LIN {X -0.032,Y -439.695,Z 1064.574,A 0.000,B 0.000,C 90.000,E1 103.300} C_DIS
LIN {X -0.146,Y -459.814,Z 1064.563,A 0.000,B 0.000,C 90.000,E1 101.299} C_DIS
LIN {X 0.195,Y -467.473,Z 1064.559,A 0.000,B 0.000,C 90.000,E1 100.546} C_DIS
LIN {X 0.213,Y -469.559,Z 1064.557,A 0.000,B 0.000,C 90.000,E1 100.310} C_DIS
LIN {X 0.062,Y -471.262,Z 1064.556,A 0.000,B 0.000,C 90.000,E1 100.074} C_DIS
LIN {X -0.172,Y -472.541,Z 1064.555,A 0.000,B 0.000,C 90.000,E1 99.849} C_DIS
LIN {X 0.011,Y -474.126,Z 1064.552,A 0.000,B 0.000,C 90.000,E1 99.321} C_DIS
LIN {X 0.125,Y -474.657,Z 1064.549,A 0.000,B 0.000,C 90.000,E1 98.803} C_DIS
LIN {X -0.219,Y -474.225,Z 1064.546,A 0.000,B 0.000,C 90.000,E1 98.341} C_DIS
LIN {X -0.024,Y -472.767,Z 1064.543,A 0.000,B 0.000,C 90.000,E1 97.814} C_DIS
LIN {X -0.227,Y -471.579,Z 1064.542,A 0.000,B 0.000,C 90.000,E1 97.587} C_DIS
LIN {X -0.105,Y -468.181,Z 1064.539,A 0.000,B 0.000,C 90.000,E1 97.068} C_DIS
LIN {X -0.042,Y -455.689,Z 1064.529,A 0.000,B 0.000,C 90.000,E1 95.277} C_DIS
LIN {X -0.126,Y -441.483,Z 1064.518,A 0.000,B 0.000,C 90.000,E1 93.212} C_DIS
LIN {X -0.111,Y -423.738,Z 1064.501,A 0.000,B 0.000,C 90.000,E1 90.286} C_DIS
LIN {X 0.172,Y -407.307,Z 1064.485,A 0.000,B 0.000,C 90.000,E1 87.249} C_DIS
LIN {X 0.158,Y -398.335,Z 1064.476,A 0.000,B 0.000,C 90.000,E1 85.584} C_DIS
LIN {X 0.025,Y -389.176,Z 1064.466,A 0.000,B 0.000,C 90.000,E1 83.913} C_DIS
LIN {X 0.131,Y -378.261,Z 1064.455,A 0.000,B 0.000,C 90.000,E1 81.894} C_DIS
LIN {X 0.126,Y -370.259,Z 1064.447,A 0.000,B 0.000,C 90.000,E1 80.443} C_DIS
LIN {X -0.030,Y -360.352,Z 1064.437,A 0.000,B 0.000,C 90.000,E1 78.701} C_DIS
LIN {X 0.062,Y -348.682,Z 1064.426,A 0.000,B 0.000,C 90.000,E1 76.589} C_DIS
LIN {X -0.132,Y -333.953,Z 1064.410,A 0.000,B 0.000,C 90.000,E1 73.866} C_DIS
LIN {X -0.123,Y -319.754,Z 1064.395,A 0.000,B 0.000,C 90.000,E1 71.040} C_DIS
LIN {X 0.015,Y -304.809,Z 1064.377,A 0.000,B 0.000,C 90.000,E1 67.794} C_DIS
LIN {X 0.035,Y -293.366,Z 1064.362,A 0.000,B 0.000,C 90.000,E1 65.153} C_DIS
LIN {X 0.087,Y -284.911,Z 1064.351,A 0.000,B 0.000,C 90.000,E1 63.127} C_DIS
LIN {X -0.007,Y -273.876,Z 1064.336,A 0.000,B 0.000,C 90.000,E1 60.411} C_DIS
LIN {X 0.165,Y -263.096,Z 1064.320,A 0.000,B 0.000,C 90.000,E1 57.582} C_DIS
LIN {X 0.021,Y -251.353,Z 1064.302,A 0.000,B 0.000,C 90.000,E1 54.402} C_DIS
LIN {X -0.006,Y -241.398,Z 1064.286,A 0.000,B 0.000,C 90.000,E1 51.492} C_DIS
LIN {X -0.088,Y -230.859,Z 1064.267,A 0.000,B 0.000,C 90.000,E1 48.162} C_DIS
LIN {X 0.020,Y -221.065,Z 1064.248,A 0.000,B 0.000,C 90.000,E1 44.717} C_DIS
LIN {X -0.019,Y -212.891,Z 1064.231,A 0.000,B 0.000,C 90.000,E1 41.634} C_DIS
LIN {X 0.064,Y -205.107,Z 1064.214,A 0.000,B 0.000,C 90.000,E1 38.463} C_DIS
LIN {X -0.106,Y -197.961,Z 1064.196,A 0.000,B 0.000,C 90.000,E1 35.311} C_DIS
LIN {X 0.082,Y -191.433,Z 1064.178,A 0.000,B 0.000,C 90.000,E1 32.005} C_DIS
LIN {X -0.035,Y -185.633,Z 1064.160,A 0.000,B 0.000,C 90.000,E1 28.743} C_DIS
LIN {X -0.062,Y -180.529,Z 1064.141,A 0.000,B 0.000,C 90.000,E1 25.412} C_DIS
LIN {X -0.037,Y -176.142,Z 1064.122,A 0.000,B 0.000,C 90.000,E1 22.025} C_DIS
LIN {X 0.006,Y -172.503,Z 1064.103,A 0.000,B 0.000,C 90.000,E1 18.598} C_DIS
LIN {X -0.017,Y -168.891,Z 1064.079,A 0.000,B 0.000,C 90.000,E1 14.300} C_DIS
LIN {X -0.035,Y -165.957,Z 1064.050,A 0.000,B 0.000,C 90.000,E1 9.095} C_DIS
LIN {X 0.021,Y -164.114,Z 1064.007,A 0.000,B 0.000,C 90.000,E1 1.203} C_DIS
LIN {X -0.010,Y -165.807,Z 1063.958,A 0.000,B 0.000,C 90.000,E1 352.527} C_DIS
LIN {X -0.018,Y -168.701,Z 1063.929,A 0.000,B 0.000,C 90.000,E1 347.297} C_DIS
LIN {X 0.004,Y -172.281,Z 1063.905,A 0.000,B 0.000,C 90.000,E1 342.960} C_DIS
LIN {X 0.023,Y -175.889,Z 1063.886,A 0.000,B 0.000,C 90.000,E1 339.518} C_DIS
LIN {X 0.053,Y -180.218,Z 1063.867,A 0.000,B 0.000,C 90.000,E1 336.102} C_DIS
LIN {X 0.009,Y -185.294,Z 1063.849,A 0.000,B 0.000,C 90.000,E1 332.743} C_DIS
LIN {X 0.012,Y -191.186,Z 1063.830,A 0.000,B 0.000,C 90.000,E1 329.410} C_DIS
LIN {X -0.034,Y -197.896,Z 1063.812,A 0.000,B 0.000,C 90.000,E1 326.135} C_DIS
LIN {X -0.009,Y -205.317,Z 1063.794,A 0.000,B 0.000,C 90.000,E1 322.889} C_DIS
LIN {X 0.047,Y -214.515,Z 1063.774,A 0.000,B 0.000,C 90.000,E1 319.299} C_DIS
LIN {X -0.076,Y -223.380,Z 1063.757,A 0.000,B 0.000,C 90.000,E1 316.215} C_DIS
LIN {X -0.097,Y -231.825,Z 1063.742,A 0.000,B 0.000,C 90.000,E1 313.542} C_DIS
LIN {X -0.099,Y -242.772,Z 1063.725,A 0.000,B 0.000,C 90.000,E1 310.539} C_DIS
LIN {X 0.024,Y -250.496,Z 1063.715,A 0.000,B 0.000,C 90.000,E1 308.669} C_DIS
LIN {X -0.007,Y -260.943,Z 1063.703,A 0.000,B 0.000,C 90.000,E1 306.503} C_DIS
LIN {X 0.163,Y -278.361,Z 1063.685,A 0.000,B 0.000,C 90.000,E1 303.293} C_DIS
LIN {X 0.013,Y -294.989,Z 1063.670,A 0.000,B 0.000,C 90.000,E1 300.590} C_DIS
LIN {X -0.175,Y -312.721,Z 1063.655,A 0.000,B 0.000,C 90.000,E1 297.975} C_DIS
LIN {X -0.152,Y -329.507,Z 1063.643,A 0.000,B 0.000,C 90.000,E1 295.720} C_DIS
LIN {X -0.105,Y -339.902,Z 1063.636,A 0.000,B 0.000,C 90.000,E1 294.463} C_DIS
LIN {X -0.113,Y -355.907,Z 1063.626,A 0.000,B 0.000,C 90.000,E1 292.770} C_DIS
LIN {X 0.102,Y -375.164,Z 1063.616,A 0.000,B 0.000,C 90.000,E1 290.918} C_DIS
LIN {X 0.090,Y -394.606,Z 1063.607,A 0.000,B 0.000,C 90.000,E1 289.214} C_DIS
LIN {X -0.133,Y -405.562,Z 1063.602,A 0.000,B 0.000,C 90.000,E1 288.308} C_DIS
LIN {X 0.077,Y -416.195,Z 1063.596,A 0.000,B 0.000,C 90.000,E1 287.330} C_DIS
LIN {X 0.042,Y -423.799,Z 1063.592,A 0.000,B 0.000,C 90.000,E1 286.622} C_DIS
LIN {X 0.136,Y -430.980,Z 1063.588,A 0.000,B 0.000,C 90.000,E1 285.898} C_DIS
LIN {X -0.129,Y -440.679,Z 1063.583,A 0.000,B 0.000,C 90.000,E1 284.898} C_DIS
LIN {X 0.191,Y -447.662,Z 1063.578,A 0.000,B 0.000,C 90.000,E1 284.064} C_DIS
LIN {X 0.035,Y -454.176,Z 1063.574,A 0.000,B 0.000,C 90.000,E1 283.300} C_DIS
LIN {X -0.074,Y -459.997,Z 1063.570,A 0.000,B 0.000,C 90.000,E1 282.535} C_DIS
LIN {X -0.127,Y -465.162,Z 1063.565,A 0.000,B 0.000,C 90.000,E1 281.771} C_DIS
LIN {X -0.143,Y -469.654,Z 1063.561,A 0.000,B 0.000,C 90.000,E1 281.007} C_DIS
LIN {X -0.205,Y -473.432,Z 1063.557,A 0.000,B 0.000,C 90.000,E1 280.254} C_DIS
LIN {X -0.233,Y -476.636,Z 1063.553,A 0.000,B 0.000,C 90.000,E1 279.500} C_DIS
LIN {X -0.026,Y -478.476,Z 1063.550,A 0.000,B 0.000,C 90.000,E1 278.973} C_DIS
LIN {X 0.114,Y -480.089,Z 1063.547,A 0.000,B 0.000,C 90.000,E1 278.454} C_DIS
LIN {X 0.017,Y -482.687,Z 1063.542,A 0.000,B 0.000,C 90.000,E1 277.466} C_DIS
LIN {X 0.187,Y -483.768,Z 1063.539,A 0.000,B 0.000,C 90.000,E1 276.947} C_DIS
LIN {X -0.116,Y -484.581,Z 1063.536,A 0.000,B 0.000,C 90.000,E1 276.486} C_DIS
LIN {X 0.067,Y -485.137,Z 1063.533,A 0.000,B 0.000,C 90.000,E1 275.967} C_DIS
LIN {X 0.209,Y -485.234,Z 1063.530,A 0.000,B 0.000,C 90.000,E1 275.454} C_DIS
LIN {X -0.080,Y -484.976,Z 1063.528,A 0.000,B 0.000,C 90.000,E1 274.992} C_DIS
LIN {X 0.112,Y -484.243,Z 1063.525,A 0.000,B 0.000,C 90.000,E1 274.473} C_DIS
LIN {X -0.181,Y -482.986,Z 1063.522,A 0.000,B 0.000,C 90.000,E1 274.012} C_DIS
LIN {X -0.031,Y -481.115,Z 1063.519,A 0.000,B 0.000,C 90.000,E1 273.498} C_DIS
LIN {X 0.141,Y -478.649,Z 1063.517,A 0.000,B 0.000,C 90.000,E1 272.980} C_DIS
LIN {X -0.206,Y -475.363,Z 1063.514,A 0.000,B 0.000,C 90.000,E1 272.522} C_DIS
LIN {X -0.089,Y -471.247,Z 1063.511,A 0.000,B 0.000,C 90.000,E1 272.007} C_DIS
LIN {X 0.020,Y -466.048,Z 1063.508,A 0.000,B 0.000,C 90.000,E1 271.489} C_DIS
LIN {X -0.096,Y -460.287,Z 1063.506,A 0.000,B 0.000,C 90.000,E1 271.031} C_DIS
LIN {X 0.167,Y -454.105,Z 1063.503,A 0.000,B 0.000,C 90.000,E1 270.573} C_DIS
LIN {X -0.046,Y -447.420,Z 1063.501,A 0.000,B 0.000,C 90.000,E1 270.229} C_DIS
LIN {X -0.220,Y -440.237,Z 1063.500,A 0.000,B 0.000,C 90.000,E1 269.943} C_DIS
LIN {X 0.089,Y -432.502,Z 1063.498,A 0.000,B 0.000,C 90.000,E1 269.656} C_DIS
LIN {X 0.000,Y -424.409,Z 1063.497,A 0.000,B 0.000,C 90.000,E1 269.484} C_DIS
LIN {X -0.129,Y -415.458,Z 1063.496,A 0.000,B 0.000,C 90.000,E1 269.370} C_DIS
LIN {X 0.032,Y -406.189,Z 1063.496,A 0.000,B 0.000,C 90.000,E1 269.255} C_DIS
LIN {X 0.039,Y -395.853,Z 1063.496,A 0.000,B 0.000,C 90.000,E1 269.198} C_DIS
LIN {X -0.012,Y -181.363,Z 1063.495,A 0.000,B 0.000,C 90.000,E1 269.198} C_DIS
LIN {X 0.045,Y -180.907,Z 1063.475,A 0.000,B 0.000,C 90.000,E1 265.469} C_DIS
LIN {X -0.078,Y -180.743,Z 1063.470,A 0.000,B 0.000,C 90.000,E1 264.666} C_DIS
LIN {X 0.023,Y -178.834,Z 1063.442,A 0.000,B 0.000,C 90.000,E1 259.567} C_DIS
LIN {X 0.057,Y -175.878,Z 1063.414,A 0.000,B 0.000,C 90.000,E1 254.464} C_DIS
LIN {X -0.006,Y -174.538,Z 1063.404,A 0.000,B 0.000,C 90.000,E1 252.779} C_DIS
LIN {X 0.087,Y -171.523,Z 1063.380,A 0.000,B 0.000,C 90.000,E1 248.465} C_DIS
LIN {X 0.072,Y -167.749,Z 1063.357,A 0.000,B 0.000,C 90.000,E1 244.152} C_DIS
LIN {X 0.011,Y -166.451,Z 1063.347,A 0.000,B 0.000,C 90.000,E1 242.436} C_DIS
LIN {X 0.001,Y -163.168,Z 1063.328,A 0.000,B 0.000,C 90.000,E1 238.948} C_DIS
LIN {X 0.050,Y -161.126,Z 1063.313,A 0.000,B 0.000,C 90.000,E1 236.294} C_DIS
LIN {X -0.047,Y -157.148,Z 1063.288,A 0.000,B 0.000,C 90.000,E1 231.904} C_DIS
LIN {X -0.024,Y -155.881,Z 1063.278,A 0.000,B 0.000,C 90.000,E1 230.114} C_DIS
LIN {X -0.065,Y -152.132,Z 1063.253,A 0.000,B 0.000,C 90.000,E1 225.648} C_DIS
LIN {X -0.045,Y -150.381,Z 1063.238,A 0.000,B 0.000,C 90.000,E1 222.933} C_DIS
LIN {X -0.021,Y -147.114,Z 1063.213,A 0.000,B 0.000,C 90.000,E1 218.382} C_DIS
LIN {X -0.029,Y -145.680,Z 1063.198,A 0.000,B 0.000,C 90.000,E1 215.644} C_DIS
LIN {X -0.031,Y -143.062,Z 1063.172,A 0.000,B 0.000,C 90.000,E1 211.052} C_DIS
LIN {X 0.026,Y -141.683,Z 1063.152,A 0.000,B 0.000,C 90.000,E1 207.334} C_DIS
LIN {X 0.005,Y -139.458,Z 1063.116,A 0.000,B 0.000,C 90.000,E1 200.844} C_DIS
LIN {X 0.056,Y -139.192,Z 1063.105,A 0.000,B 0.000,C 90.000,E1 198.960} C_DIS
LIN {X -0.057,Y -138.325,Z 1063.054,A 0.000,B 0.000,C 90.000,E1 189.670} C_DIS
LIN {X -0.053,Y -139.455,Z 1063.007,A 0.000,B 0.000,C 90.000,E1 181.260} C_DIS
LIN {X 0.027,Y -141.003,Z 1062.976,A 0.000,B 0.000,C 90.000,E1 175.641} C_DIS
LIN {X -0.023,Y -142.757,Z 1062.955,A 0.000,B 0.000,C 90.000,E1 171.951} C_DIS
LIN {X -0.068,Y -145.160,Z 1062.930,A 0.000,B 0.000,C 90.000,E1 167.353} C_DIS
LIN {X -0.076,Y -147.782,Z 1062.909,A 0.000,B 0.000,C 90.000,E1 163.685} C_DIS
LIN {X 0.003,Y -150.461,Z 1062.889,A 0.000,B 0.000,C 90.000,E1 160.007} C_DIS
LIN {X 0.079,Y -153.912,Z 1062.869,A 0.000,B 0.000,C 90.000,E1 156.357} C_DIS
LIN {X 0.003,Y -157.323,Z 1062.849,A 0.000,B 0.000,C 90.000,E1 152.794} C_DIS
LIN {X 0.087,Y -161.511,Z 1062.829,A 0.000,B 0.000,C 90.000,E1 149.203} C_DIS
LIN {X -0.036,Y -165.710,Z 1062.809,A 0.000,B 0.000,C 90.000,E1 145.722} C_DIS
LIN {X 0.089,Y -170.656,Z 1062.790,A 0.000,B 0.000,C 90.000,E1 142.190} C_DIS
LIN {X 0.002,Y -175.533,Z 1062.771,A 0.000,B 0.000,C 90.000,E1 138.771} C_DIS
LIN {X -0.004,Y -181.152,Z 1062.752,A 0.000,B 0.000,C 90.000,E1 135.364} C_DIS
LIN {X -0.007,Y -186.605,Z 1062.733,A 0.000,B 0.000,C 90.000,E1 132.000} C_DIS
LIN {X 0.063,Y -191.214,Z 1062.719,A 0.000,B 0.000,C 90.000,E1 129.483} C_DIS
LIN {X -0.009,Y -197.425,Z 1062.700,A 0.000,B 0.000,C 90.000,E1 126.011} C_DIS
LIN {X -0.052,Y -198.581,Z 1062.697,A 0.000,B 0.000,C 90.000,E1 125.438} C_DIS
LIN {X -0.114,Y -305.000,Z 1062.697,A 0.000,B 0.000,C 90.000,E1 125.438} C_DIS
LIN {X 0.033,Y -306.362,Z 1062.697,A 0.000,B 0.000,C 90.000,E1 125.391} C_DIS
LIN {X -0.186,Y -309.700,Z 1062.696,A 0.000,B 0.000,C 90.000,E1 125.311} C_DIS
LIN {X 0.137,Y -312.965,Z 1062.695,A 0.000,B 0.000,C 90.000,E1 125.025} C_DIS
LIN {X 0.124,Y -316.653,Z 1062.692,A 0.000,B 0.000,C 90.000,E1 124.612} C_DIS
LIN {X 0.011,Y -318.561,Z 1062.691,A 0.000,B 0.000,C 90.000,E1 124.326} C_DIS
LIN {X 0.161,Y -320.060,Z 1062.689,A 0.000,B 0.000,C 90.000,E1 123.992} C_DIS
LIN {X -0.136,Y -323.460,Z 1062.684,A 0.000,B 0.000,C 90.000,E1 123.086} C_DIS
LIN {X 0.070,Y -333.960,Z 1062.668,A 0.000,B 0.000,C 90.000,E1 120.207} C_DIS
LIN {X -0.043,Y -345.811,Z 1062.652,A 0.000,B 0.000,C 90.000,E1 117.436} C_DIS
LIN {X -0.005,Y -359.122,Z 1062.637,A 0.000,B 0.000,C 90.000,E1 114.695} C_DIS
LIN {X -0.119,Y -372.270,Z 1062.624,A 0.000,B 0.000,C 90.000,E1 112.333} C_DIS
LIN {X -0.042,Y -386.756,Z 1062.611,A 0.000,B 0.000,C 90.000,E1 109.993} C_DIS
LIN {X 0.138,Y -402.680,Z 1062.598,A 0.000,B 0.000,C 90.000,E1 107.692} C_DIS
LIN {X 0.088,Y -420.157,Z 1062.586,A 0.000,B 0.000,C 90.000,E1 105.481} C_DIS
LIN {X -0.155,Y -439.292,Z 1062.574,A 0.000,B 0.000,C 90.000,E1 103.355} C_DIS
LIN {X 0.146,Y -459.401,Z 1062.563,A 0.000,B 0.000,C 90.000,E1 101.299} C_DIS
LIN {X 0.023,Y -467.071,Z 1062.559,A 0.000,B 0.000,C 90.000,E1 100.602} C_DIS
LIN {X 0.036,Y -469.257,Z 1062.558,A 0.000,B 0.000,C 90.000,E1 100.366} C_DIS
LIN {X -0.199,Y -471.030,Z 1062.556,A 0.000,B 0.000,C 90.000,E1 100.141} C_DIS
LIN {X 0.113,Y -472.363,Z 1062.555,A 0.000,B 0.000,C 90.000,E1 99.849} C_DIS
LIN {X -0.172,Y -474.028,Z 1062.552,A 0.000,B 0.000,C 90.000,E1 99.378} C_DIS
LIN {X -0.062,Y -474.628,Z 1062.549,A 0.000,B 0.000,C 90.000,E1 98.859} C_DIS
LIN {X 0.063,Y -474.263,Z 1062.546,A 0.000,B 0.000,C 90.000,E1 98.341} C_DIS
LIN {X -0.211,Y -472.881,Z 1062.544,A 0.000,B 0.000,C 90.000,E1 97.871} C_DIS
LIN {X 0.054,Y -471.740,Z 1062.542,A 0.000,B 0.000,C 90.000,E1 97.587} C_DIS
LIN {X -0.085,Y -470.219,Z 1062.541,A 0.000,B 0.000,C 90.000,E1 97.352} C_DIS
LIN {X 0.234,Y -455.909,Z 1062.530,A 0.000,B 0.000,C 90.000,E1 95.277} C_DIS
LIN {X -0.091,Y -440.013,Z 1062.516,A 0.000,B 0.000,C 90.000,E1 92.980} C_DIS
LIN {X -0.018,Y -420.855,Z 1062.499,A 0.000,B 0.000,C 90.000,E1 89.771} C_DIS
LIN {X 0.029,Y -407.518,Z 1062.485,A 0.000,B 0.000,C 90.000,E1 87.306} C_DIS
LIN {X 0.023,Y -398.552,Z 1062.476,A 0.000,B 0.000,C 90.000,E1 85.641} C_DIS
LIN {X -0.102,Y -389.400,Z 1062.466,A 0.000,B 0.000,C 90.000,E1 83.970} C_DIS
LIN {X 0.014,Y -378.487,Z 1062.455,A 0.000,B 0.000,C 90.000,E1 81.951} C_DIS
LIN {X 0.016,Y -370.516,Z 1062.447,A 0.000,B 0.000,C 90.000,E1 80.500} C_DIS
LIN {X -0.131,Y -360.565,Z 1062.437,A 0.000,B 0.000,C 90.000,E1 78.757} C_DIS
LIN {X -0.029,Y -348.903,Z 1062.426,A 0.000,B 0.000,C 90.000,E1 76.645} C_DIS
LIN {X 0.113,Y -334.198,Z 1062.411,A 0.000,B 0.000,C 90.000,E1 73.866} C_DIS
LIN {X 0.117,Y -319.964,Z 1062.395,A 0.000,B 0.000,C 90.000,E1 71.040} C_DIS
LIN {X -0.032,Y -305.005,Z 1062.377,A 0.000,B 0.000,C 90.000,E1 67.847} C_DIS
LIN {X -0.124,Y -293.541,Z 1062.362,A 0.000,B 0.000,C 90.000,E1 65.229} C_DIS
LIN {X -0.092,Y -283.663,Z 1062.349,A 0.000,B 0.000,C 90.000,E1 62.871} C_DIS
LIN {X -0.077,Y -272.652,Z 1062.334,A 0.000,B 0.000,C 90.000,E1 60.127} C_DIS
LIN {X -0.066,Y -261.880,Z 1062.318,A 0.000,B 0.000,C 90.000,E1 57.327} C_DIS
LIN {X -0.099,Y -250.180,Z 1062.301,A 0.000,B 0.000,C 90.000,E1 54.116} C_DIS
LIN {X -0.001,Y -240.219,Z 1062.284,A 0.000,B 0.000,C 90.000,E1 51.170} C_DIS
LIN {X 0.067,Y -229.739,Z 1062.266,A 0.000,B 0.000,C 90.000,E1 47.796} C_DIS
LIN {X 0.053,Y -221.070,Z 1062.249,A 0.000,B 0.000,C 90.000,E1 44.757} C_DIS
LIN {X 0.003,Y -212.870,Z 1062.232,A 0.000,B 0.000,C 90.000,E1 41.676} C_DIS
LIN {X -0.051,Y -205.075,Z 1062.214,A 0.000,B 0.000,C 90.000,E1 38.543} C_DIS
LIN {X 0.060,Y -197.919,Z 1062.196,A 0.000,B 0.000,C 90.000,E1 35.311} C_DIS
LIN {X -0.021,Y -191.371,Z 1062.178,A 0.000,B 0.000,C 90.000,E1 32.084} C_DIS
LIN {X 0.030,Y -185.550,Z 1062.160,A 0.000,B 0.000,C 90.000,E1 28.771} C_DIS
LIN {X -0.078,Y -180.434,Z 1062.141,A 0.000,B 0.000,C 90.000,E1 25.463} C_DIS
LIN {X -0.059,Y -176.029,Z 1062.123,A 0.000,B 0.000,C 90.000,E1 22.078} C_DIS
LIN {X -0.022,Y -172.389,Z 1062.104,A 0.000,B 0.000,C 90.000,E1 18.652} C_DIS
LIN {X -0.051,Y -168.752,Z 1062.080,A 0.000,B 0.000,C 90.000,E1 14.356} C_DIS
LIN {X -0.062,Y -166.194,Z 1062.056,A 0.000,B 0.000,C 90.000,E1 10.018} C_DIS
LIN {X 0.067,Y -164.072,Z 1062.017,A 0.000,B 0.000,C 90.000,E1 2.980} C_DIS
LIN {X 0.004,Y -165.293,Z 1061.963,A 0.000,B 0.000,C 90.000,E1 353.394} C_DIS
LIN {X -0.048,Y -167.974,Z 1061.934,A 0.000,B 0.000,C 90.000,E1 348.173} C_DIS
LIN {X 0.073,Y -171.333,Z 1061.910,A 0.000,B 0.000,C 90.000,E1 343.795} C_DIS
LIN {X 0.017,Y -174.773,Z 1061.891,A 0.000,B 0.000,C 90.000,E1 340.369} C_DIS
LIN {X -0.049,Y -178.917,Z 1061.872,A 0.000,B 0.000,C 90.000,E1 336.975} C_DIS
LIN {X -0.040,Y -183.833,Z 1061.853,A 0.000,B 0.000,C 90.000,E1 333.589} C_DIS
LIN {X -0.076,Y -189.535,Z 1061.835,A 0.000,B 0.000,C 90.000,E1 330.255} C_DIS
LIN {X 0.062,Y -196.027,Z 1061.816,A 0.000,B 0.000,C 90.000,E1 326.914} C_DIS
LIN {X -0.082,Y -203.297,Z 1061.798,A 0.000,B 0.000,C 90.000,E1 323.703} C_DIS
LIN {X 0.004,Y -211.273,Z 1061.780,A 0.000,B 0.000,C 90.000,E1 320.481} C_DIS
LIN {X 0.131,Y -219.857,Z 1061.763,A 0.000,B 0.000,C 90.000,E1 317.310} C_DIS
LIN {X -0.025,Y -229.199,Z 1061.746,A 0.000,B 0.000,C 90.000,E1 314.271} C_DIS
LIN {X 0.070,Y -239.800,Z 1061.729,A 0.000,B 0.000,C 90.000,E1 311.229} C_DIS
LIN {X -0.040,Y -247.155,Z 1061.719,A 0.000,B 0.000,C 90.000,E1 309.402} C_DIS
LIN {X -0.139,Y -257.230,Z 1061.707,A 0.000,B 0.000,C 90.000,E1 307.237} C_DIS
LIN {X 0.080,Y -270.354,Z 1061.693,A 0.000,B 0.000,C 90.000,E1 304.692} C_DIS
LIN {X 0.000,Y -288.580,Z 1061.676,A 0.000,B 0.000,C 90.000,E1 301.592} C_DIS
LIN {X 0.064,Y -305.895,Z 1061.661,A 0.000,B 0.000,C 90.000,E1 298.899} C_DIS
LIN {X 0.100,Y -327.053,Z 1061.644,A 0.000,B 0.000,C 90.000,E1 295.976} C_DIS
LIN {X -0.186,Y -340.026,Z 1061.636,A 0.000,B 0.000,C 90.000,E1 294.463} C_DIS
LIN {X -0.037,Y -353.504,Z 1061.628,A 0.000,B 0.000,C 90.000,E1 293.003} C_DIS
LIN {X -0.079,Y -372.970,Z 1061.617,A 0.000,B 0.000,C 90.000,E1 291.153} C_DIS
LIN {X -0.145,Y -392.379,Z 1061.608,A 0.000,B 0.000,C 90.000,E1 289.450} C_DIS
LIN {X 0.071,Y -406.153,Z 1061.601,A 0.000,B 0.000,C 90.000,E1 288.236} C_DIS
LIN {X 0.119,Y -416.781,Z 1061.596,A 0.000,B 0.000,C 90.000,E1 287.275} C_DIS
LIN {X 0.011,Y -424.440,Z 1061.592,A 0.000,B 0.000,C 90.000,E1 286.567} C_DIS
LIN {X -0.179,Y -431.921,Z 1061.588,A 0.000,B 0.000,C 90.000,E1 285.843} C_DIS
LIN {X 0.008,Y -441.656,Z 1061.582,A 0.000,B 0.000,C 90.000,E1 284.773} C_DIS
LIN {X -0.211,Y -448.606,Z 1061.578,A 0.000,B 0.000,C 90.000,E1 284.008} C_DIS
LIN {X 0.183,Y -454.997,Z 1061.573,A 0.000,B 0.000,C 90.000,E1 283.175} C_DIS
LIN {X 0.081,Y -460.728,Z 1061.569,A 0.000,B 0.000,C 90.000,E1 282.411} C_DIS
LIN {X -0.063,Y -465.811,Z 1061.565,A 0.000,B 0.000,C 90.000,E1 281.658} C_DIS
LIN {X -0.071,Y -470.235,Z 1061.560,A 0.000,B 0.000,C 90.000,E1 280.894} C_DIS
LIN {X -0.124,Y -473.954,Z 1061.556,A 0.000,B 0.000,C 90.000,E1 280.141} C_DIS
LIN {X -0.066,Y -477.123,Z 1061.552,A 0.000,B 0.000,C 90.000,E1 279.378} C_DIS
LIN {X 0.068,Y -478.914,Z 1061.549,A 0.000,B 0.000,C 90.000,E1 278.859} C_DIS
LIN {X 0.212,Y -480.495,Z 1061.547,A 0.000,B 0.000,C 90.000,E1 278.341} C_DIS
LIN {X 0.122,Y -483.081,Z 1061.541,A 0.000,B 0.000,C 90.000,E1 277.352} C_DIS
LIN {X -0.185,Y -484.106,Z 1061.538,A 0.000,B 0.000,C 90.000,E1 276.891} C_DIS
LIN {X -0.005,Y -484.903,Z 1061.535,A 0.000,B 0.000,C 90.000,E1 276.372} C_DIS
LIN {X 0.182,Y -485.384,Z 1061.533,A 0.000,B 0.000,C 90.000,E1 275.853} C_DIS
LIN {X -0.111,Y -485.441,Z 1061.530,A 0.000,B 0.000,C 90.000,E1 275.391} C_DIS
LIN {X 0.041,Y -485.093,Z 1061.527,A 0.000,B 0.000,C 90.000,E1 274.878} C_DIS
LIN {X 0.234,Y -484.238,Z 1061.524,A 0.000,B 0.000,C 90.000,E1 274.359} C_DIS
LIN {X -0.059,Y -482.885,Z 1061.522,A 0.000,B 0.000,C 90.000,E1 273.898} C_DIS
LIN {X 0.092,Y -480.924,Z 1061.519,A 0.000,B 0.000,C 90.000,E1 273.383} C_DIS
LIN {X -0.214,Y -478.285,Z 1061.516,A 0.000,B 0.000,C 90.000,E1 272.922} C_DIS
LIN {X -0.086,Y -474.868,Z 1061.513,A 0.000,B 0.000,C 90.000,E1 272.407} C_DIS
LIN {X 0.028,Y -470.537,Z 1061.510,A 0.000,B 0.000,C 90.000,E1 271.892} C_DIS
LIN {X 0.131,Y -465.160,Z 1061.508,A 0.000,B 0.000,C 90.000,E1 271.375} C_DIS
LIN {X 0.093,Y -459.290,Z 1061.505,A 0.000,B 0.000,C 90.000,E1 270.917} C_DIS
LIN {X -0.030,Y -453.038,Z 1061.503,A 0.000,B 0.000,C 90.000,E1 270.516} C_DIS
LIN {X -0.146,Y -446.382,Z 1061.501,A 0.000,B 0.000,C 90.000,E1 270.172} C_DIS
LIN {X 0.184,Y -439.078,Z 1061.499,A 0.000,B 0.000,C 90.000,E1 269.828} C_DIS
LIN {X 0.145,Y -435.601,Z 1061.499,A 0.000,B 0.000,C 90.000,E1 269.714} C_DIS
LIN {X -0.086,Y -427.543,Z 1061.497,A 0.000,B 0.000,C 90.000,E1 269.542} C_DIS
LIN {X 0.110,Y -419.418,Z 1061.497,A 0.000,B 0.000,C 90.000,E1 269.370} C_DIS
LIN {X 0.168,Y -410.058,Z 1061.496,A 0.000,B 0.000,C 90.000,E1 269.255} C_DIS
LIN {X -0.054,Y -395.709,Z 1061.495,A 0.000,B 0.000,C 90.000,E1 269.198} C_DIS
LIN {X -0.053,Y -181.361,Z 1061.495,A 0.000,B 0.000,C 90.000,E1 269.198} C_DIS
LIN {X -0.023,Y -180.907,Z 1061.475,A 0.000,B 0.000,C 90.000,E1 265.469} C_DIS
LIN {X 0.034,Y -180.733,Z 1061.470,A 0.000,B 0.000,C 90.000,E1 264.609} C_DIS
LIN {X -0.045,Y -178.823,Z 1061.442,A 0.000,B 0.000,C 90.000,E1 259.567} C_DIS
LIN {X 0.037,Y -175.867,Z 1061.414,A 0.000,B 0.000,C 90.000,E1 254.448} C_DIS
LIN {X 0.032,Y -173.837,Z 1061.399,A 0.000,B 0.000,C 90.000,E1 251.891} C_DIS
LIN {X 0.020,Y -171.504,Z 1061.380,A 0.000,B 0.000,C 90.000,E1 248.465} C_DIS
LIN {X 0.007,Y -167.733,Z 1061.356,A 0.000,B 0.000,C 90.000,E1 244.152} C_DIS
LIN {X 0.022,Y -166.429,Z 1061.347,A 0.000,B 0.000,C 90.000,E1 242.410} C_DIS
LIN {X 0.021,Y -163.149,Z 1061.327,A 0.000,B 0.000,C 90.000,E1 238.918} C_DIS
LIN {X -0.013,Y -161.105,Z 1061.313,A 0.000,B 0.000,C 90.000,E1 236.294} C_DIS
LIN {X -0.030,Y -157.831,Z 1061.293,A 0.000,B 0.000,C 90.000,E1 232.763} C_DIS
LIN {X 0.033,Y -155.864,Z 1061.278,A 0.000,B 0.000,C 90.000,E1 230.070} C_DIS
LIN {X 0.088,Y -152.114,Z 1061.253,A 0.000,B 0.000,C 90.000,E1 225.567} C_DIS
LIN {X -0.004,Y -150.365,Z 1061.238,A 0.000,B 0.000,C 90.000,E1 222.894} C_DIS
LIN {X 0.035,Y -147.100,Z 1061.213,A 0.000,B 0.000,C 90.000,E1 218.338} C_DIS
LIN {X 0.029,Y -145.669,Z 1061.198,A 0.000,B 0.000,C 90.000,E1 215.598} C_DIS
LIN {X 0.032,Y -143.050,Z 1061.172,A 0.000,B 0.000,C 90.000,E1 211.003} C_DIS
LIN {X -0.033,Y -141.673,Z 1061.152,A 0.000,B 0.000,C 90.000,E1 207.334} C_DIS
LIN {X 0.076,Y -139.454,Z 1061.116,A 0.000,B 0.000,C 90.000,E1 200.791} C_DIS
LIN {X -0.003,Y -139.188,Z 1061.105,A 0.000,B 0.000,C 90.000,E1 198.960} C_DIS
LIN {X 0.020,Y -138.323,Z 1061.053,A 0.000,B 0.000,C 90.000,E1 189.613} C_DIS
LIN {X 0.027,Y -139.458,Z 1061.007,A 0.000,B 0.000,C 90.000,E1 181.203} C_DIS
LIN {X -0.032,Y -141.012,Z 1060.976,A 0.000,B 0.000,C 90.000,E1 175.641} C_DIS
LIN {X 0.058,Y -142.766,Z 1060.955,A 0.000,B 0.000,C 90.000,E1 171.894} C_DIS
LIN {X 0.013,Y -145.175,Z 1060.929,A 0.000,B 0.000,C 90.000,E1 167.297} C_DIS
LIN {X 0.047,Y -147.797,Z 1060.909,A 0.000,B 0.000,C 90.000,E1 163.614} C_DIS
LIN {X -0.058,Y -150.482,Z 1060.889,A 0.000,B 0.000,C 90.000,E1 160.007} C_DIS
LIN {X 0.016,Y -153.935,Z 1060.869,A 0.000,B 0.000,C 90.000,E1 156.357} C_DIS
LIN {X 0.078,Y -157.347,Z 1060.849,A 0.000,B 0.000,C 90.000,E1 152.743} C_DIS
LIN {X 0.022,Y -161.542,Z 1060.829,A 0.000,B 0.000,C 90.000,E1 149.203} C_DIS
LIN {X 0.035,Y -165.740,Z 1060.809,A 0.000,B 0.000,C 90.000,E1 145.674} C_DIS
LIN {X 0.023,Y -170.692,Z 1060.790,A 0.000,B 0.000,C 90.000,E1 142.190} C_DIS
LIN {X -0.066,Y -175.566,Z 1060.771,A 0.000,B 0.000,C 90.000,E1 138.771} C_DIS
LIN {X 0.054,Y -181.184,Z 1060.752,A 0.000,B 0.000,C 90.000,E1 135.324} C_DIS
LIN {X -0.078,Y -186.643,Z 1060.733,A 0.000,B 0.000,C 90.000,E1 132.000} C_DIS
LIN {X -0.008,Y -191.249,Z 1060.719,A 0.000,B 0.000,C 90.000,E1 129.483} C_DIS
LIN {X -0.075,Y -197.462,Z 1060.700,A 0.000,B 0.000,C 90.000,E1 126.011} C_DIS
LIN {X -0.014,Y -198.492,Z 1060.697,A 0.000,B 0.000,C 90.000,E1 125.471} C_DIS
LIN {X 0.120,Y -304.825,Z 1060.697,A 0.000,B 0.000,C 90.000,E1 125.438} C_DIS
LIN {X -0.080,Y -308.346,Z 1060.697,A 0.000,B 0.000,C 90.000,E1 125.391} C_DIS
LIN {X -0.061,Y -311.200,Z 1060.696,A 0.000,B 0.000,C 90.000,E1 125.231} C_DIS
LIN {X -0.074,Y -314.877,Z 1060.694,A 0.000,B 0.000,C 90.000,E1 124.898} C_DIS
LIN {X 0.022,Y -318.448,Z 1060.691,A 0.000,B 0.000,C 90.000,E1 124.358} C_DIS
LIN {X 0.002,Y -320.002,Z 1060.689,A 0.000,B 0.000,C 90.000,E1 124.040} C_DIS
LIN {X 0.047,Y -324.482,Z 1060.682,A 0.000,B 0.000,C 90.000,E1 122.752} C_DIS
LIN {X 0.002,Y -335.120,Z 1060.666,A 0.000,B 0.000,C 90.000,E1 119.922} C_DIS
LIN {X 0.057,Y -347.119,Z 1060.651,A 0.000,B 0.000,C 90.000,E1 117.129} C_DIS
LIN {X 0.144,Y -360.588,Z 1060.636,A 0.000,B 0.000,C 90.000,E1 114.387} C_DIS
LIN {X 0.076,Y -373.891,Z 1060.622,A 0.000,B 0.000,C 90.000,E1 112.025} C_DIS
LIN {X 0.070,Y -388.541,Z 1060.609,A 0.000,B 0.000,C 90.000,E1 109.704} C_DIS
LIN {X -0.075,Y -404.642,Z 1060.597,A 0.000,B 0.000,C 90.000,E1 107.457} C_DIS
LIN {X -0.082,Y -422.311,Z 1060.585,A 0.000,B 0.000,C 90.000,E1 105.245} C_DIS
LIN {X 0.178,Y -441.619,Z 1060.573,A 0.000,B 0.000,C 90.000,E1 103.063} C_DIS
LIN {X 0.119,Y -461.796,Z 1060.562,A 0.000,B 0.000,C 90.000,E1 101.074} C_DIS
LIN {X 0.108,Y -466.926,Z 1060.559,A 0.000,B 0.000,C 90.000,E1 100.602} C_DIS
LIN {X 0.142,Y -469.124,Z 1060.558,A 0.000,B 0.000,C 90.000,E1 100.366} C_DIS
LIN {X 0.091,Y -470.786,Z 1060.556,A 0.000,B 0.000,C 90.000,E1 100.141} C_DIS
LIN {X -0.055,Y -472.170,Z 1060.555,A 0.000,B 0.000,C 90.000,E1 99.905} C_DIS
LIN {X -0.202,Y -473.197,Z 1060.554,A 0.000,B 0.000,C 90.000,E1 99.670} C_DIS
LIN {X -0.094,Y -474.381,Z 1060.551,A 0.000,B 0.000,C 90.000,E1 99.151} C_DIS
LIN {X 0.098,Y -474.564,Z 1060.548,A 0.000,B 0.000,C 90.000,E1 98.624} C_DIS
LIN {X 0.223,Y -473.781,Z 1060.545,A 0.000,B 0.000,C 90.000,E1 98.106} C_DIS
LIN {X -0.118,Y -471.903,Z 1060.542,A 0.000,B 0.000,C 90.000,E1 97.644} C_DIS
LIN {X 0.208,Y -470.442,Z 1060.541,A 0.000,B 0.000,C 90.000,E1 97.352} C_DIS
LIN {X -0.199,Y -457.944,Z 1060.531,A 0.000,B 0.000,C 90.000,E1 95.625} C_DIS
LIN {X 0.200,Y -440.234,Z 1060.517,A 0.000,B 0.000,C 90.000,E1 92.980} C_DIS
LIN {X -0.039,Y -419.550,Z 1060.497,A 0.000,B 0.000,C 90.000,E1 89.542} C_DIS
LIN {X -0.026,Y -406.258,Z 1060.484,A 0.000,B 0.000,C 90.000,E1 87.078} C_DIS
LIN {X 0.009,Y -395.759,Z 1060.473,A 0.000,B 0.000,C 90.000,E1 85.122} C_DIS
LIN {X -0.163,Y -386.522,Z 1060.464,A 0.000,B 0.000,C 90.000,E1 83.451} C_DIS
LIN {X -0.121,Y -377.158,Z 1060.454,A 0.000,B 0.000,C 90.000,E1 81.724} C_DIS
LIN {X -0.141,Y -369.103,Z 1060.446,A 0.000,B 0.000,C 90.000,E1 80.274} C_DIS
LIN {X 0.068,Y -357.457,Z 1060.434,A 0.000,B 0.000,C 90.000,E1 78.173} C_DIS
LIN {X 0.100,Y -345.817,Z 1060.423,A 0.000,B 0.000,C 90.000,E1 76.061} C_DIS
LIN {X -0.086,Y -331.212,Z 1060.407,A 0.000,B 0.000,C 90.000,E1 73.323} C_DIS
LIN {X 0.014,Y -318.647,Z 1060.393,A 0.000,B 0.000,C 90.000,E1 70.786} C_DIS
LIN {X -0.063,Y -305.226,Z 1060.377,A 0.000,B 0.000,C 90.000,E1 67.901} C_DIS
LIN {X -0.009,Y -292.315,Z 1060.361,A 0.000,B 0.000,C 90.000,E1 64.921} C_DIS
LIN {X -0.012,Y -282.424,Z 1060.348,A 0.000,B 0.000,C 90.000,E1 62.564} C_DIS
LIN {X 0.098,Y -271.451,Z 1060.332,A 0.000,B 0.000,C 90.000,E1 59.793} C_DIS
LIN {X -0.060,Y -262.004,Z 1060.319,A 0.000,B 0.000,C 90.000,E1 57.375} C_DIS
LIN {X 0.126,Y -250.280,Z 1060.301,A 0.000,B 0.000,C 90.000,E1 54.116} C_DIS
LIN {X -0.120,Y -240.282,Z 1060.285,A 0.000,B 0.000,C 90.000,E1 51.251} C_DIS
LIN {X -0.051,Y -229.772,Z 1060.266,A 0.000,B 0.000,C 90.000,E1 47.877} C_DIS
LIN {X 0.020,Y -220.044,Z 1060.247,A 0.000,B 0.000,C 90.000,E1 44.433} C_DIS
LIN {X 0.103,Y -211.867,Z 1060.230,A 0.000,B 0.000,C 90.000,E1 41.310} C_DIS
LIN {X 0.025,Y -204.136,Z 1060.212,A 0.000,B 0.000,C 90.000,E1 38.177} C_DIS
LIN {X -0.006,Y -197.028,Z 1060.194,A 0.000,B 0.000,C 90.000,E1 34.978} C_DIS
LIN {X -0.003,Y -190.555,Z 1060.176,A 0.000,B 0.000,C 90.000,E1 31.720} C_DIS
LIN {X 0.018,Y -184.791,Z 1060.158,A 0.000,B 0.000,C 90.000,E1 28.409} C_DIS
LIN {X -0.035,Y -179.759,Z 1060.139,A 0.000,B 0.000,C 90.000,E1 25.079} C_DIS
LIN {X 0.061,Y -175.432,Z 1060.120,A 0.000,B 0.000,C 90.000,E1 21.663} C_DIS
LIN {X 0.086,Y -171.856,Z 1060.101,A 0.000,B 0.000,C 90.000,E1 18.236} C_DIS
LIN {X -0.001,Y -168.311,Z 1060.078,A 0.000,B 0.000,C 90.000,E1 13.953} C_DIS
LIN {X -0.035,Y -165.483,Z 1060.048,A 0.000,B 0.000,C 90.000,E1 8.746} C_DIS
LIN {X 0.000,Y -163.800,Z 1060.000,A 0.000,B 0.000,C 90.000,E1 360.000} C_DIS
LIN {X -0.026,Y -165.502,Z 1059.958,A 0.000,B 0.000,C 90.000,E1 352.527} C_DIS
LIN {X -0.007,Y -168.424,Z 1059.929,A 0.000,B 0.000,C 90.000,E1 347.285} C_DIS
LIN {X -0.032,Y -171.959,Z 1059.905,A 0.000,B 0.000,C 90.000,E1 342.960} C_DIS
LIN {X -0.021,Y -175.602,Z 1059.886,A 0.000,B 0.000,C 90.000,E1 339.518} C_DIS
LIN {X 0.000,Y -179.951,Z 1059.867,A 0.000,B 0.000,C 90.000,E1 336.102} C_DIS
LIN {X -0.052,Y -185.065,Z 1059.849,A 0.000,B 0.000,C 90.000,E1 332.743} C_DIS
LIN {X -0.056,Y -190.971,Z 1059.830,A 0.000,B 0.000,C 90.000,E1 329.410} C_DIS
LIN {X 0.054,Y -197.700,Z 1059.812,A 0.000,B 0.000,C 90.000,E1 326.087} C_DIS
LIN {X -0.051,Y -206.070,Z 1059.792,A 0.000,B 0.000,C 90.000,E1 322.477} C_DIS
LIN {X -0.141,Y -215.390,Z 1059.772,A 0.000,B 0.000,C 90.000,E1 318.933} C_DIS
LIN {X -0.015,Y -225.475,Z 1059.752,A 0.000,B 0.000,C 90.000,E1 315.405} C_DIS
LIN {X -0.147,Y -234.231,Z 1059.737,A 0.000,B 0.000,C 90.000,E1 312.771} C_DIS
LIN {X 0.128,Y -242.516,Z 1059.725,A 0.000,B 0.000,C 90.000,E1 310.458} C_DIS
LIN {X -0.099,Y -250.243,Z 1059.715,A 0.000,B 0.000,C 90.000,E1 308.669} C_DIS
LIN {X 0.070,Y -260.722,Z 1059.703,A 0.000,B 0.000,C 90.000,E1 306.457} C_DIS
LIN {X 0.015,Y -278.201,Z 1059.685,A 0.000,B 0.000,C 90.000,E1 303.293} C_DIS
LIN {X 0.106,Y -294.878,Z 1059.670,A 0.000,B 0.000,C 90.000,E1 300.541} C_DIS
LIN {X -0.023,Y -315.075,Z 1059.653,A 0.000,B 0.000,C 90.000,E1 297.590} C_DIS
LIN {X -0.035,Y -329.619,Z 1059.643,A 0.000,B 0.000,C 90.000,E1 295.668} C_DIS
LIN {X 0.162,Y -340.161,Z 1059.636,A 0.000,B 0.000,C 90.000,E1 294.387} C_DIS
LIN {X -0.087,Y -353.635,Z 1059.628,A 0.000,B 0.000,C 90.000,E1 293.003} C_DIS
LIN {X 0.046,Y -372.631,Z 1059.618,A 0.000,B 0.000,C 90.000,E1 291.173} C_DIS
LIN {X 0.196,Y -391.907,Z 1059.608,A 0.000,B 0.000,C 90.000,E1 289.450} C_DIS
LIN {X -0.086,Y -402.931,Z 1059.603,A 0.000,B 0.000,C 90.000,E1 288.544} C_DIS
LIN {X -0.007,Y -411.071,Z 1059.599,A 0.000,B 0.000,C 90.000,E1 287.819} C_DIS
LIN {X 0.028,Y -418.955,Z 1059.595,A 0.000,B 0.000,C 90.000,E1 287.094} C_DIS
LIN {X -0.127,Y -426.671,Z 1059.591,A 0.000,B 0.000,C 90.000,E1 286.370} C_DIS
LIN {X 0.096,Y -436.566,Z 1059.585,A 0.000,B 0.000,C 90.000,E1 285.315} C_DIS
LIN {X 0.013,Y -443.795,Z 1059.581,A 0.000,B 0.000,C 90.000,E1 284.537} C_DIS
LIN {X -0.179,Y -450.557,Z 1059.576,A 0.000,B 0.000,C 90.000,E1 283.772} C_DIS
LIN {X 0.123,Y -456.786,Z 1059.572,A 0.000,B 0.000,C 90.000,E1 282.952} C_DIS
LIN {X 0.048,Y -462.299,Z 1059.568,A 0.000,B 0.000,C 90.000,E1 282.187} C_DIS
LIN {X 0.011,Y -467.236,Z 1059.563,A 0.000,B 0.000,C 90.000,E1 281.422} C_DIS
LIN {X 0.019,Y -471.452,Z 1059.559,A 0.000,B 0.000,C 90.000,E1 280.658} C_DIS
LIN {X -0.028,Y -475.031,Z 1059.555,A 0.000,B 0.000,C 90.000,E1 279.905} C_DIS
LIN {X 0.171,Y -477.088,Z 1059.552,A 0.000,B 0.000,C 90.000,E1 279.378} C_DIS
LIN {X -0.168,Y -478.902,Z 1059.549,A 0.000,B 0.000,C 90.000,E1 278.916} C_DIS
LIN {X -0.026,Y -480.525,Z 1059.547,A 0.000,B 0.000,C 90.000,E1 278.398} C_DIS
LIN {X -0.118,Y -483.152,Z 1059.541,A 0.000,B 0.000,C 90.000,E1 277.409} C_DIS
LIN {X 0.056,Y -484.216,Z 1059.538,A 0.000,B 0.000,C 90.000,E1 276.891} C_DIS
LIN {X 0.237,Y -485.040,Z 1059.536,A 0.000,B 0.000,C 90.000,E1 276.372} C_DIS
LIN {X -0.058,Y -485.523,Z 1059.533,A 0.000,B 0.000,C 90.000,E1 275.910} C_DIS
LIN {X 0.133,Y -485.651,Z 1059.530,A 0.000,B 0.000,C 90.000,E1 275.391} C_DIS
LIN {X -0.199,Y -485.307,Z 1059.527,A 0.000,B 0.000,C 90.000,E1 274.935} C_DIS
LIN {X -0.004,Y -484.496,Z 1059.525,A 0.000,B 0.000,C 90.000,E1 274.416} C_DIS
LIN {X 0.186,Y -483.200,Z 1059.522,A 0.000,B 0.000,C 90.000,E1 273.898} C_DIS
LIN {X -0.142,Y -481.272,Z 1059.519,A 0.000,B 0.000,C 90.000,E1 273.440} C_DIS
LIN {X 0.031,Y -478.706,Z 1059.516,A 0.000,B 0.000,C 90.000,E1 272.922} C_DIS
LIN {X 0.161,Y -475.329,Z 1059.513,A 0.000,B 0.000,C 90.000,E1 272.407} C_DIS
LIN {X -0.019,Y -473.333,Z 1059.512,A 0.000,B 0.000,C 90.000,E1 272.178} C_DIS
LIN {X 0.100,Y -468.511,Z 1059.509,A 0.000,B 0.000,C 90.000,E1 271.661} C_DIS
LIN {X -0.132,Y -462.926,Z 1059.507,A 0.000,B 0.000,C 90.000,E1 271.203} C_DIS
LIN {X -0.024,Y -456.931,Z 1059.504,A 0.000,B 0.000,C 90.000,E1 270.745} C_DIS
LIN {X 0.030,Y -450.532,Z 1059.502,A 0.000,B 0.000,C 90.000,E1 270.344} C_DIS
LIN {X 0.086,Y -443.587,Z 1059.500,A 0.000,B 0.000,C 90.000,E1 270.000} C_DIS
LIN {X 0.168,Y -436.293,Z 1059.499,A 0.000,B 0.000,C 90.000,E1 269.714} C_DIS
LIN {X -0.127,Y -428.069,Z 1059.497,A 0.000,B 0.000,C 90.000,E1 269.542} C_DIS
LIN {X 0.032,Y -419.621,Z 1059.497,A 0.000,B 0.000,C 90.000,E1 269.370} C_DIS
LIN {X 0.072,Y -410.230,Z 1059.496,A 0.000,B 0.000,C 90.000,E1 269.255} C_DIS
LIN {X -0.093,Y -397.772,Z 1059.495,A 0.000,B 0.000,C 90.000,E1 269.198} C_DIS
LIN {X -0.153,Y -394.636,Z 1059.495,A 0.000,B 0.000,C 90.000,E1 269.198} C_DIS
LIN {X 0.084,Y -181.357,Z 1059.495,A 0.000,B 0.000,C 90.000,E1 269.141} C_DIS
LIN {X -0.066,Y -180.907,Z 1059.475,A 0.000,B 0.000,C 90.000,E1 265.469} C_DIS
LIN {X -0.009,Y -180.726,Z 1059.470,A 0.000,B 0.000,C 90.000,E1 264.609} C_DIS
LIN {X 0.088,Y -178.815,Z 1059.442,A 0.000,B 0.000,C 90.000,E1 259.511} C_DIS
LIN {X -0.005,Y -175.861,Z 1059.414,A 0.000,B 0.000,C 90.000,E1 254.448} C_DIS
LIN {X 0.043,Y -173.827,Z 1059.399,A 0.000,B 0.000,C 90.000,E1 251.873} C_DIS
LIN {X -0.021,Y -171.494,Z 1059.380,A 0.000,B 0.000,C 90.000,E1 248.465} C_DIS
LIN {X -0.034,Y -167.721,Z 1059.356,A 0.000,B 0.000,C 90.000,E1 244.152} C_DIS
LIN {X -0.018,Y -166.415,Z 1059.347,A 0.000,B 0.000,C 90.000,E1 242.410} C_DIS
LIN {X -0.019,Y -163.137,Z 1059.327,A 0.000,B 0.000,C 90.000,E1 238.918} C_DIS
LIN {X -0.054,Y -161.091,Z 1059.313,A 0.000,B 0.000,C 90.000,E1 236.294} C_DIS
LIN {X -0.070,Y -157.820,Z 1059.293,A 0.000,B 0.000,C 90.000,E1 232.763} C_DIS
LIN {X -0.006,Y -155.854,Z 1059.278,A 0.000,B 0.000,C 90.000,E1 230.070} C_DIS
LIN {X 0.050,Y -152.104,Z 1059.253,A 0.000,B 0.000,C 90.000,E1 225.567} C_DIS
LIN {X 0.068,Y -150.355,Z 1059.238,A 0.000,B 0.000,C 90.000,E1 222.852} C_DIS
LIN {X -0.003,Y -147.091,Z 1059.213,A 0.000,B 0.000,C 90.000,E1 218.338} C_DIS
LIN {X -0.009,Y -145.662,Z 1059.198,A 0.000,B 0.000,C 90.000,E1 215.598} C_DIS
LIN {X -0.005,Y -143.044,Z 1059.172,A 0.000,B 0.000,C 90.000,E1 211.003} C_DIS
LIN {X -0.005,Y -141.668,Z 1059.152,A 0.000,B 0.000,C 90.000,E1 207.308} C_DIS
LIN {X 0.040,Y -139.451,Z 1059.116,A 0.000,B 0.000,C 90.000,E1 200.791} C_DIS
LIN {X -0.039,Y -139.185,Z 1059.105,A 0.000,B 0.000,C 90.000,E1 198.960} C_DIS
LIN {X -0.016,Y -138.322,Z 1059.053,A 0.000,B 0.000,C 90.000,E1 189.613} C_DIS
LIN {X -0.009,Y -139.462,Z 1059.007,A 0.000,B 0.000,C 90.000,E1 181.203} C_DIS
LIN {X -0.069,Y -141.019,Z 1058.976,A 0.000,B 0.000,C 90.000,E1 175.641} C_DIS
LIN {X 0.027,Y -142.382,Z 1058.960,A 0.000,B 0.000,C 90.000,E1 172.818} C_DIS
LIN {X -0.052,Y -144.613,Z 1058.934,A 0.000,B 0.000,C 90.000,E1 168.229} C_DIS
LIN {X 0.010,Y -147.807,Z 1058.909,A 0.000,B 0.000,C 90.000,E1 163.614} C_DIS
LIN {X 0.045,Y -150.494,Z 1058.889,A 0.000,B 0.000,C 90.000,E1 159.953} C_DIS
LIN {X -0.024,Y -153.950,Z 1058.869,A 0.000,B 0.000,C 90.000,E1 156.357} C_DIS
LIN {X 0.039,Y -157.362,Z 1058.849,A 0.000,B 0.000,C 90.000,E1 152.743} C_DIS
LIN {X -0.018,Y -161.560,Z 1058.829,A 0.000,B 0.000,C 90.000,E1 149.203} C_DIS
LIN {X -0.006,Y -165.758,Z 1058.809,A 0.000,B 0.000,C 90.000,E1 145.674} C_DIS
LIN {X -0.019,Y -170.713,Z 1058.790,A 0.000,B 0.000,C 90.000,E1 142.190} C_DIS
LIN {X 0.024,Y -175.586,Z 1058.771,A 0.000,B 0.000,C 90.000,E1 138.728} C_DIS
LIN {X 0.011,Y -181.204,Z 1058.752,A 0.000,B 0.000,C 90.000,E1 135.324} C_DIS
LIN {X 0.004,Y -186.668,Z 1058.733,A 0.000,B 0.000,C 90.000,E1 131.962} C_DIS
LIN {X -0.052,Y -191.271,Z 1058.719,A 0.000,B 0.000,C 90.000,E1 129.483} C_DIS
LIN {X 0.043,Y -197.485,Z 1058.700,A 0.000,B 0.000,C 90.000,E1 125.964} C_DIS
LIN {X -0.027,Y -198.406,Z 1058.697,A 0.000,B 0.000,C 90.000,E1 125.518} C_DIS
LIN {X -0.076,Y -304.369,Z 1058.697,A 0.000,B 0.000,C 90.000,E1 125.518} C_DIS
LIN {X -0.151,Y -309.372,Z 1058.696,A 0.000,B 0.000,C 90.000,E1 125.391} C_DIS
LIN {X -0.002,Y -312.075,Z 1058.695,A 0.000,B 0.000,C 90.000,E1 125.185} C_DIS
LIN {X -0.181,Y -315.856,Z 1058.693,A 0.000,B 0.000,C 90.000,E1 124.818} C_DIS
LIN {X 0.048,Y -317.786,Z 1058.692,A 0.000,B 0.000,C 90.000,E1 124.485} C_DIS
LIN {X 0.016,Y -319.310,Z 1058.690,A 0.000,B 0.000,C 90.000,E1 124.199} C_DIS
LIN {X 0.090,Y -320.638,Z 1058.688,A 0.000,B 0.000,C 90.000,E1 123.865} C_DIS
LIN {X -0.053,Y -332.000,Z 1058.671,A 0.000,B 0.000,C 90.000,E1 120.718} C_DIS
LIN {X 0.068,Y -343.610,Z 1058.655,A 0.000,B 0.000,C 90.000,E1 117.897} C_DIS
LIN {X 0.057,Y -356.657,Z 1058.640,A 0.000,B 0.000,C 90.000,E1 115.155} C_DIS
LIN {X 0.038,Y -369.555,Z 1058.627,A 0.000,B 0.000,C 90.000,E1 112.770} C_DIS
LIN {X 0.055,Y -383.770,Z 1058.614,A 0.000,B 0.000,C 90.000,E1 110.429} C_DIS
LIN {X -0.209,Y -399.404,Z 1058.601,A 0.000,B 0.000,C 90.000,E1 108.181} C_DIS
LIN {X 0.169,Y -416.568,Z 1058.589,A 0.000,B 0.000,C 90.000,E1 105.898} C_DIS
LIN {X -0.173,Y -435.385,Z 1058.576,A 0.000,B 0.000,C 90.000,E1 103.772} C_DIS
LIN {X -0.142,Y -455.379,Z 1058.565,A 0.000,B 0.000,C 90.000,E1 101.715} C_DIS
LIN {X 0.080,Y -468.081,Z 1058.558,A 0.000,B 0.000,C 90.000,E1 100.489} C_DIS
LIN {X 0.049,Y -470.040,Z 1058.557,A 0.000,B 0.000,C 90.000,E1 100.254} C_DIS
LIN {X 0.018,Y -471.527,Z 1058.556,A 0.000,B 0.000,C 90.000,E1 100.018} C_DIS
LIN {X -0.127,Y -472.716,Z 1058.554,A 0.000,B 0.000,C 90.000,E1 99.782} C_DIS
LIN {X 0.114,Y -473.582,Z 1058.553,A 0.000,B 0.000,C 90.000,E1 99.500} C_DIS
LIN {X -0.164,Y -474.496,Z 1058.550,A 0.000,B 0.000,C 90.000,E1 99.029} C_DIS
LIN {X -0.046,Y -474.432,Z 1058.547,A 0.000,B 0.000,C 90.000,E1 98.511} C_DIS
LIN {X 0.082,Y -473.386,Z 1058.544,A 0.000,B 0.000,C 90.000,E1 97.992} C_DIS
LIN {X -0.056,Y -472.447,Z 1058.543,A 0.000,B 0.000,C 90.000,E1 97.757} C_DIS
LIN {X -0.258,Y -471.176,Z 1058.542,A 0.000,B 0.000,C 90.000,E1 97.530} C_DIS
LIN {X 0.091,Y -460.580,Z 1058.533,A 0.000,B 0.000,C 90.000,E1 95.967} C_DIS
LIN {X 0.151,Y -449.810,Z 1058.525,A 0.000,B 0.000,C 90.000,E1 94.416} C_DIS
LIN {X 0.199,Y -437.687,Z 1058.515,A 0.000,B 0.000,C 90.000,E1 92.579} C_DIS
LIN {X -0.122,Y -417.256,Z 1058.495,A 0.000,B 0.000,C 90.000,E1 89.141} C_DIS
LIN {X 0.168,Y -405.494,Z 1058.483,A 0.000,B 0.000,C 90.000,E1 86.906} C_DIS
LIN {X 0.181,Y -394.994,Z 1058.472,A 0.000,B 0.000,C 90.000,E1 84.951} C_DIS
LIN {X -0.011,Y -385.735,Z 1058.463,A 0.000,B 0.000,C 90.000,E1 83.280} C_DIS
LIN {X 0.078,Y -374.756,Z 1058.451,A 0.000,B 0.000,C 90.000,E1 81.254} C_DIS
LIN {X 0.020,Y -366.577,Z 1058.443,A 0.000,B 0.000,C 90.000,E1 79.803} C_DIS
LIN {X 0.181,Y -354.920,Z 1058.432,A 0.000,B 0.000,C 90.000,E1 77.701} C_DIS
LIN {X 0.155,Y -341.669,Z 1058.418,A 0.000,B 0.000,C 90.000,E1 75.283} C_DIS
LIN {X -0.003,Y -328.789,Z 1058.405,A 0.000,B 0.000,C 90.000,E1 72.834} C_DIS
LIN {X -0.132,Y -314.824,Z 1058.389,A 0.000,B 0.000,C 90.000,E1 70.007} C_DIS
LIN {X -0.102,Y -302.994,Z 1058.374,A 0.000,B 0.000,C 90.000,E1 67.411} C_DIS
LIN {X 0.145,Y -291.560,Z 1058.360,A 0.000,B 0.000,C 90.000,E1 64.717} C_DIS
LIN {X 0.087,Y -280.288,Z 1058.345,A 0.000,B 0.000,C 90.000,E1 62.025} C_DIS
LIN {X 0.012,Y -269.344,Z 1058.329,A 0.000,B 0.000,C 90.000,E1 59.282} C_DIS
LIN {X -0.148,Y -258.594,Z 1058.314,A 0.000,B 0.000,C 90.000,E1 56.501} C_DIS
LIN {X 0.082,Y -247.032,Z 1058.296,A 0.000,B 0.000,C 90.000,E1 53.210} C_DIS
LIN {X 0.029,Y -235.976,Z 1058.277,A 0.000,B 0.000,C 90.000,E1 49.908} C_DIS
LIN {X -0.041,Y -225.745,Z 1058.259,A 0.000,B 0.000,C 90.000,E1 46.539} C_DIS
LIN {X 0.017,Y -217.298,Z 1058.241,A 0.000,B 0.000,C 90.000,E1 43.461} C_DIS
LIN {X 0.048,Y -209.222,Z 1058.224,A 0.000,B 0.000,C 90.000,E1 40.334} C_DIS
LIN {X 0.065,Y -201.705,Z 1058.207,A 0.000,B 0.000,C 90.000,E1 37.156} C_DIS
LIN {X 0.130,Y -194.754,Z 1058.189,A 0.000,B 0.000,C 90.000,E1 33.913} C_DIS
LIN {X 0.027,Y -188.526,Z 1058.170,A 0.000,B 0.000,C 90.000,E1 30.669} C_DIS
LIN {X -0.086,Y -182.952,Z 1058.152,A 0.000,B 0.000,C 90.000,E1 27.385} C_DIS
LIN {X -0.019,Y -178.150,Z 1058.133,A 0.000,B 0.000,C 90.000,E1 24.003} C_DIS
LIN {X -0.031,Y -174.050,Z 1058.115,A 0.000,B 0.000,C 90.000,E1 20.610} C_DIS
LIN {X -0.019,Y -169.949,Z 1058.091,A 0.000,B 0.000,C 90.000,E1 16.315} C_DIS
LIN {X -0.083,Y -166.854,Z 1058.067,A 0.000,B 0.000,C 90.000,E1 12.007} C_DIS
LIN {X 0.045,Y -164.323,Z 1058.033,A 0.000,B 0.000,C 90.000,E1 5.853} C_DIS
LIN {X -0.034,Y -165.358,Z 1057.958,A 0.000,B 0.000,C 90.000,E1 352.527} C_DIS
LIN {X -0.020,Y -168.287,Z 1057.929,A 0.000,B 0.000,C 90.000,E1 347.285} C_DIS
LIN {X -0.050,Y -171.823,Z 1057.905,A 0.000,B 0.000,C 90.000,E1 342.960} C_DIS
LIN {X -0.042,Y -175.480,Z 1057.886,A 0.000,B 0.000,C 90.000,E1 339.518} C_DIS
LIN {X -0.025,Y -179.830,Z 1057.867,A 0.000,B 0.000,C 90.000,E1 336.102} C_DIS
LIN {X -0.080,Y -184.948,Z 1057.848,A 0.000,B 0.000,C 90.000,E1 332.743} C_DIS
LIN {X -0.088,Y -190.874,Z 1057.830,A 0.000,B 0.000,C 90.000,E1 329.410} C_DIS
LIN {X -0.010,Y -195.821,Z 1057.816,A 0.000,B 0.000,C 90.000,E1 326.914} C_DIS
LIN {X 0.123,Y -203.090,Z 1057.798,A 0.000,B 0.000,C 90.000,E1 323.623} C_DIS
LIN {X 0.086,Y -211.079,Z 1057.780,A 0.000,B 0.000,C 90.000,E1 320.436} C_DIS
LIN {X -0.043,Y -220.804,Z 1057.761,A 0.000,B 0.000,C 90.000,E1 316.944} C_DIS
LIN {X -0.024,Y -230.245,Z 1057.744,A 0.000,B 0.000,C 90.000,E1 313.866} C_DIS
LIN {X -0.038,Y -239.544,Z 1057.729,A 0.000,B 0.000,C 90.000,E1 311.229} C_DIS
LIN {X 0.036,Y -246.923,Z 1057.719,A 0.000,B 0.000,C 90.000,E1 309.358} C_DIS
LIN {X 0.055,Y -253.490,Z 1057.711,A 0.000,B 0.000,C 90.000,E1 307.890} C_DIS
LIN {X -0.020,Y -266.273,Z 1057.697,A 0.000,B 0.000,C 90.000,E1 305.391} C_DIS
LIN {X -0.070,Y -284.310,Z 1057.679,A 0.000,B 0.000,C 90.000,E1 302.260} C_DIS
LIN {X 0.029,Y -303.661,Z 1057.662,A 0.000,B 0.000,C 90.000,E1 299.205} C_DIS
LIN {X -0.005,Y -324.686,Z 1057.646,A 0.000,B 0.000,C 90.000,E1 296.283} C_DIS
LIN {X -0.104,Y -337.616,Z 1057.637,A 0.000,B 0.000,C 90.000,E1 294.719} C_DIS
LIN {X 0.104,Y -350.859,Z 1057.629,A 0.000,B 0.000,C 90.000,E1 293.259} C_DIS
LIN {X -0.197,Y -372.561,Z 1057.618,A 0.000,B 0.000,C 90.000,E1 291.227} C_DIS
LIN {X -0.095,Y -391.889,Z 1057.608,A 0.000,B 0.000,C 90.000,E1 289.504} C_DIS
LIN {X -0.001,Y -405.609,Z 1057.602,A 0.000,B 0.000,C 90.000,E1 288.308} C_DIS
LIN {X -0.238,Y -416.115,Z 1057.596,A 0.000,B 0.000,C 90.000,E1 287.402} C_DIS
LIN {X 0.090,Y -423.861,Z 1057.592,A 0.000,B 0.000,C 90.000,E1 286.622} C_DIS
LIN {X -0.190,Y -431.419,Z 1057.588,A 0.000,B 0.000,C 90.000,E1 285.898} C_DIS
LIN {X -0.017,Y -441.224,Z 1057.582,A 0.000,B 0.000,C 90.000,E1 284.828} C_DIS
LIN {X -0.234,Y -448.172,Z 1057.578,A 0.000,B 0.000,C 90.000,E1 284.064} C_DIS
LIN {X 0.051,Y -454.587,Z 1057.574,A 0.000,B 0.000,C 90.000,E1 283.244} C_DIS
LIN {X -0.052,Y -460.354,Z 1057.569,A 0.000,B 0.000,C 90.000,E1 282.479} C_DIS
LIN {X -0.101,Y -465.494,Z 1057.565,A 0.000,B 0.000,C 90.000,E1 281.715} C_DIS
LIN {X -0.112,Y -470.023,Z 1057.561,A 0.000,B 0.000,C 90.000,E1 280.950} C_DIS
LIN {X -0.170,Y -473.842,Z 1057.557,A 0.000,B 0.000,C 90.000,E1 280.197} C_DIS
LIN {X -0.115,Y -477.072,Z 1057.552,A 0.000,B 0.000,C 90.000,E1 279.434} C_DIS
LIN {X 0.161,Y -480.543,Z 1057.547,A 0.000,B 0.000,C 90.000,E1 278.398} C_DIS
LIN {X -0.160,Y -482.003,Z 1057.544,A 0.000,B 0.000,C 90.000,E1 277.936} C_DIS
LIN {X 0.069,Y -483.261,Z 1057.541,A 0.000,B 0.000,C 90.000,E1 277.409} C_DIS
LIN {X 0.243,Y -484.340,Z 1057.538,A 0.000,B 0.000,C 90.000,E1 276.891} C_DIS
LIN {X -0.056,Y -485.147,Z 1057.536,A 0.000,B 0.000,C 90.000,E1 276.429} C_DIS
LIN {X 0.131,Y -485.662,Z 1057.533,A 0.000,B 0.000,C 90.000,E1 275.910} C_DIS
LIN {X -0.160,Y -485.808,Z 1057.530,A 0.000,B 0.000,C 90.000,E1 275.448} C_DIS
LIN {X -0.008,Y -485.490,Z 1057.527,A 0.000,B 0.000,C 90.000,E1 274.935} C_DIS
LIN {X 0.187,Y -484.741,Z 1057.525,A 0.000,B 0.000,C 90.000,E1 274.416} C_DIS
LIN {X -0.104,Y -483.449,Z 1057.522,A 0.000,B 0.000,C 90.000,E1 273.955} C_DIS
LIN {X 0.050,Y -481.568,Z 1057.519,A 0.000,B 0.000,C 90.000,E1 273.440} C_DIS
LIN {X 0.224,Y -479.062,Z 1057.516,A 0.000,B 0.000,C 90.000,E1 272.922} C_DIS
LIN {X -0.120,Y -475.712,Z 1057.514,A 0.000,B 0.000,C 90.000,E1 272.465} C_DIS
LIN {X -0.002,Y -471.514,Z 1057.511,A 0.000,B 0.000,C 90.000,E1 271.949} C_DIS
LIN {X 0.107,Y -466.267,Z 1057.508,A 0.000,B 0.000,C 90.000,E1 271.432} C_DIS
LIN {X 0.004,Y -460.471,Z 1057.505,A 0.000,B 0.000,C 90.000,E1 270.974} C_DIS
LIN {X -0.199,Y -454.246,Z 1057.503,A 0.000,B 0.000,C 90.000,E1 270.573} C_DIS
LIN {X 0.004,Y -447.542,Z 1057.501,A 0.000,B 0.000,C 90.000,E1 270.172} C_DIS
LIN {X -0.186,Y -440.322,Z 1057.499,A 0.000,B 0.000,C 90.000,E1 269.885} C_DIS
LIN {X 0.175,Y -436.833,Z 1057.499,A 0.000,B 0.000,C 90.000,E1 269.714} C_DIS
LIN {X -0.151,Y -428.717,Z 1057.497,A 0.000,B 0.000,C 90.000,E1 269.542} C_DIS
LIN {X -0.015,Y -420.090,Z 1057.496,A 0.000,B 0.000,C 90.000,E1 269.370} C_DIS
LIN {X 0.009,Y -410.816,Z 1057.496,A 0.000,B 0.000,C 90.000,E1 269.255} C_DIS
LIN {X -0.167,Y -397.785,Z 1057.495,A 0.000,B 0.000,C 90.000,E1 269.198} C_DIS
LIN {X 0.169,Y -394.655,Z 1057.495,A 0.000,B 0.000,C 90.000,E1 269.141} C_DIS
LIN {X 0.050,Y -181.355,Z 1057.495,A 0.000,B 0.000,C 90.000,E1 269.141} C_DIS
LIN {X 0.081,Y -180.906,Z 1057.475,A 0.000,B 0.000,C 90.000,E1 265.412} C_DIS
LIN {X -0.043,Y -180.723,Z 1057.470,A 0.000,B 0.000,C 90.000,E1 264.609} C_DIS
LIN {X 0.056,Y -178.810,Z 1057.442,A 0.000,B 0.000,C 90.000,E1 259.511} C_DIS
LIN {X -0.038,Y -175.855,Z 1057.414,A 0.000,B 0.000,C 90.000,E1 254.448} C_DIS
LIN {X -0.056,Y -173.182,Z 1057.395,A 0.000,B 0.000,C 90.000,E1 251.040} C_DIS
LIN {X -0.053,Y -171.484,Z 1057.380,A 0.000,B 0.000,C 90.000,E1 248.465} C_DIS
LIN {X -0.066,Y -167.713,Z 1057.356,A 0.000,B 0.000,C 90.000,E1 244.152} C_DIS
LIN {X -0.049,Y -166.404,Z 1057.347,A 0.000,B 0.000,C 90.000,E1 242.410} C_DIS
LIN {X 0.089,Y -163.128,Z 1057.327,A 0.000,B 0.000,C 90.000,E1 238.869} C_DIS
LIN {X -0.085,Y -161.080,Z 1057.313,A 0.000,B 0.000,C 90.000,E1 236.294} C_DIS
LIN {X 0.026,Y -157.810,Z 1057.293,A 0.000,B 0.000,C 90.000,E1 232.718} C_DIS
LIN {X -0.036,Y -155.845,Z 1057.278,A 0.000,B 0.000,C 90.000,E1 230.070} C_DIS
LIN {X 0.020,Y -152.096,Z 1057.253,A 0.000,B 0.000,C 90.000,E1 225.567} C_DIS
LIN {X 0.039,Y -150.347,Z 1057.238,A 0.000,B 0.000,C 90.000,E1 222.852} C_DIS
LIN {X 0.059,Y -147.084,Z 1057.213,A 0.000,B 0.000,C 90.000,E1 218.302} C_DIS
LIN {X -0.037,Y -145.657,Z 1057.198,A 0.000,B 0.000,C 90.000,E1 215.598} C_DIS
LIN {X -0.033,Y -143.038,Z 1057.172,A 0.000,B 0.000,C 90.000,E1 211.003} C_DIS
LIN {X -0.033,Y -141.664,Z 1057.152,A 0.000,B 0.000,C 90.000,E1 207.308} C_DIS
LIN {X 0.012,Y -139.449,Z 1057.115,A 0.000,B 0.000,C 90.000,E1 200.791} C_DIS
LIN {X 0.064,Y -139.182,Z 1057.105,A 0.000,B 0.000,C 90.000,E1 198.906} C_DIS
LIN {X -0.044,Y -138.321,Z 1057.053,A 0.000,B 0.000,C 90.000,E1 189.613} C_DIS
LIN {X -0.037,Y -139.463,Z 1057.007,A 0.000,B 0.000,C 90.000,E1 181.203} C_DIS
LIN {X 0.043,Y -141.023,Z 1056.976,A 0.000,B 0.000,C 90.000,E1 175.584} C_DIS
LIN {X -0.003,Y -142.388,Z 1056.960,A 0.000,B 0.000,C 90.000,E1 172.818} C_DIS
LIN {X 0.060,Y -144.620,Z 1056.934,A 0.000,B 0.000,C 90.000,E1 168.173} C_DIS
LIN {X -0.020,Y -147.814,Z 1056.909,A 0.000,B 0.000,C 90.000,E1 163.614} C_DIS
LIN {X 0.067,Y -150.503,Z 1056.889,A 0.000,B 0.000,C 90.000,E1 159.934} C_DIS
LIN {X -0.053,Y -153.962,Z 1056.869,A 0.000,B 0.000,C 90.000,E1 156.357} C_DIS
LIN {X 0.009,Y -157.373,Z 1056.849,A 0.000,B 0.000,C 90.000,E1 152.743} C_DIS
LIN {X -0.049,Y -161.575,Z 1056.829,A 0.000,B 0.000,C 90.000,E1 149.203} C_DIS
LIN {X -0.038,Y -165.772,Z 1056.809,A 0.000,B 0.000,C 90.000,E1 145.674} C_DIS
LIN {X -0.051,Y -170.730,Z 1056.790,A 0.000,B 0.000,C 90.000,E1 142.190} C_DIS
LIN {X -0.009,Y -175.603,Z 1056.771,A 0.000,B 0.000,C 90.000,E1 138.728} C_DIS
LIN {X -0.023,Y -181.220,Z 1056.752,A 0.000,B 0.000,C 90.000,E1 135.324} C_DIS
LIN {X -0.030,Y -186.686,Z 1056.733,A 0.000,B 0.000,C 90.000,E1 131.962} C_DIS
LIN {X 0.061,Y -191.288,Z 1056.719,A 0.000,B 0.000,C 90.000,E1 129.439} C_DIS
LIN {X 0.011,Y -197.504,Z 1056.700,A 0.000,B 0.000,C 90.000,E1 125.964} C_DIS
LIN {X 0.106,Y -198.331,Z 1056.698,A 0.000,B 0.000,C 90.000,E1 125.518} C_DIS
LIN {X 0.127,Y -304.584,Z 1056.698,A 0.000,B 0.000,C 90.000,E1 125.518} C_DIS
LIN {X 0.022,Y -305.945,Z 1056.697,A 0.000,B 0.000,C 90.000,E1 125.518} C_DIS
LIN {X -0.026,Y -310.100,Z 1056.696,A 0.000,B 0.000,C 90.000,E1 125.358} C_DIS
LIN {X -0.031,Y -313.321,Z 1056.695,A 0.000,B 0.000,C 90.000,E1 125.105} C_DIS
LIN {X 0.131,Y -317.015,Z 1056.692,A 0.000,B 0.000,C 90.000,E1 124.612} C_DIS
LIN {X -0.073,Y -318.818,Z 1056.691,A 0.000,B 0.000,C 90.000,E1 124.326} C_DIS
LIN {X -0.015,Y -320.228,Z 1056.689,A 0.000,B 0.000,C 90.000,E1 123.992} C_DIS
LIN {X -0.061,Y -332.784,Z 1056.669,A 0.000,B 0.000,C 90.000,E1 120.512} C_DIS
LIN {X -0.082,Y -344.497,Z 1056.654,A 0.000,B 0.000,C 90.000,E1 117.719} C_DIS
LIN {X 0.087,Y -357.652,Z 1056.639,A 0.000,B 0.000,C 90.000,E1 114.951} C_DIS
LIN {X -0.058,Y -370.656,Z 1056.625,A 0.000,B 0.000,C 90.000,E1 112.589} C_DIS
LIN {X -0.013,Y -384.985,Z 1056.612,A 0.000,B 0.000,C 90.000,E1 110.248} C_DIS
LIN {X 0.132,Y -400.741,Z 1056.600,A 0.000,B 0.000,C 90.000,E1 107.946} C_DIS
LIN {X 0.159,Y -418.036,Z 1056.587,A 0.000,B 0.000,C 90.000,E1 105.717} C_DIS
LIN {X -0.140,Y -436.984,Z 1056.575,A 0.000,B 0.000,C 90.000,E1 103.592} C_DIS
LIN {X 0.003,Y -457.028,Z 1056.564,A 0.000,B 0.000,C 90.000,E1 101.535} C_DIS
LIN {X -0.183,Y -467.252,Z 1056.559,A 0.000,B 0.000,C 90.000,E1 100.602} C_DIS
LIN {X -0.169,Y -469.371,Z 1056.557,A 0.000,B 0.000,C 90.000,E1 100.366} C_DIS
LIN {X 0.142,Y -471.098,Z 1056.556,A 0.000,B 0.000,C 90.000,E1 100.074} C_DIS
LIN {X -0.091,Y -472.395,Z 1056.555,A 0.000,B 0.000,C 90.000,E1 99.849} C_DIS
LIN {X 0.090,Y -474.007,Z 1056.552,A 0.000,B 0.000,C 90.000,E1 99.321} C_DIS
LIN {X 0.202,Y -474.563,Z 1056.549,A 0.000,B 0.000,C 90.000,E1 98.803} C_DIS
LIN {X -0.142,Y -474.154,Z 1056.546,A 0.000,B 0.000,C 90.000,E1 98.341} C_DIS
LIN {X 0.052,Y -472.723,Z 1056.543,A 0.000,B 0.000,C 90.000,E1 97.814} C_DIS
LIN {X -0.151,Y -471.551,Z 1056.542,A 0.000,B 0.000,C 90.000,E1 97.587} C_DIS
LIN {X -0.031,Y -468.190,Z 1056.539,A 0.000,B 0.000,C 90.000,E1 97.068} C_DIS
LIN {X 0.032,Y -455.733,Z 1056.529,A 0.000,B 0.000,C 90.000,E1 95.277} C_DIS
LIN {X 0.148,Y -439.803,Z 1056.516,A 0.000,B 0.000,C 90.000,E1 92.922} C_DIS
LIN {X 0.203,Y -420.671,Z 1056.499,A 0.000,B 0.000,C 90.000,E1 89.714} C_DIS
LIN {X -0.168,Y -407.415,Z 1056.485,A 0.000,B 0.000,C 90.000,E1 87.306} C_DIS
LIN {X -0.171,Y -398.445,Z 1056.476,A 0.000,B 0.000,C 90.000,E1 85.641} C_DIS
LIN {X 0.093,Y -389.271,Z 1056.466,A 0.000,B 0.000,C 90.000,E1 83.913} C_DIS
LIN {X -0.175,Y -378.383,Z 1056.455,A 0.000,B 0.000,C 90.000,E1 81.951} C_DIS
LIN {X 0.196,Y -370.351,Z 1056.447,A 0.000,B 0.000,C 90.000,E1 80.443} C_DIS
LIN {X 0.039,Y -360.368,Z 1056.437,A 0.000,B 0.000,C 90.000,E1 78.701} C_DIS
LIN {X 0.128,Y -348.715,Z 1056.426,A 0.000,B 0.000,C 90.000,E1 76.589} C_DIS
LIN {X 0.039,Y -335.617,Z 1056.412,A 0.000,B 0.000,C 90.000,E1 74.157} C_DIS
LIN {X 0.144,Y -322.933,Z 1056.398,A 0.000,B 0.000,C 90.000,E1 71.638} C_DIS
LIN {X 0.062,Y -309.295,Z 1056.382,A 0.000,B 0.000,C 90.000,E1 68.773} C_DIS
LIN {X -0.047,Y -296.200,Z 1056.366,A 0.000,B 0.000,C 90.000,E1 65.845} C_DIS
LIN {X -0.080,Y -286.270,Z 1056.353,A 0.000,B 0.000,C 90.000,E1 63.512} C_DIS
LIN {X -0.133,Y -275.143,Z 1056.338,A 0.000,B 0.000,C 90.000,E1 60.795} C_DIS
LIN {X 0.018,Y -265.623,Z 1056.324,A 0.000,B 0.000,C 90.000,E1 58.329} C_DIS
LIN {X 0.012,Y -253.664,Z 1056.306,A 0.000,B 0.000,C 90.000,E1 55.135} C_DIS
LIN {X -0.012,Y -244.778,Z 1056.292,A 0.000,B 0.000,C 90.000,E1 52.603} C_DIS
LIN {X -0.111,Y -233.839,Z 1056.274,A 0.000,B 0.000,C 90.000,E1 49.299} C_DIS
LIN {X -0.019,Y -224.846,Z 1056.257,A 0.000,B 0.000,C 90.000,E1 46.257} C_DIS
LIN {X 0.026,Y -216.439,Z 1056.240,A 0.000,B 0.000,C 90.000,E1 43.176} C_DIS
LIN {X -0.119,Y -208.401,Z 1056.223,A 0.000,B 0.000,C 90.000,E1 40.092} C_DIS
LIN {X 0.038,Y -200.939,Z 1056.205,A 0.000,B 0.000,C 90.000,E1 36.870} C_DIS
LIN {X -0.024,Y -194.006,Z 1056.187,A 0.000,B 0.000,C 90.000,E1 33.658} C_DIS
LIN {X -0.039,Y -187.837,Z 1056.169,A 0.000,B 0.000,C 90.000,E1 30.384} C_DIS
LIN {X -0.011,Y -182.318,Z 1056.150,A 0.000,B 0.000,C 90.000,E1 27.052} C_DIS
LIN {X -0.039,Y -177.583,Z 1056.132,A 0.000,B 0.000,C 90.000,E1 23.695} C_DIS
LIN {X -0.062,Y -173.539,Z 1056.113,A 0.000,B 0.000,C 90.000,E1 20.301} C_DIS
LIN {X 0.046,Y -169.512,Z 1056.089,A 0.000,B 0.000,C 90.000,E1 15.969} C_DIS
LIN {X -0.025,Y -166.489,Z 1056.065,A 0.000,B 0.000,C 90.000,E1 11.658} C_DIS
LIN {X 0.071,Y -164.074,Z 1056.031,A 0.000,B 0.000,C 90.000,E1 5.511} C_DIS
LIN {X -0.016,Y -164.879,Z 1055.963,A 0.000,B 0.000,C 90.000,E1 353.394} C_DIS
LIN {X -0.084,Y -167.554,Z 1055.934,A 0.000,B 0.000,C 90.000,E1 348.173} C_DIS
LIN {X 0.023,Y -170.907,Z 1055.910,A 0.000,B 0.000,C 90.000,E1 343.795} C_DIS
LIN {X -0.044,Y -174.359,Z 1055.891,A 0.000,B 0.000,C 90.000,E1 340.369} C_DIS
LIN {X 0.044,Y -178.560,Z 1055.872,A 0.000,B 0.000,C 90.000,E1 336.922} C_DIS
LIN {X -0.041,Y -183.487,Z 1055.853,A 0.000,B 0.000,C 90.000,E1 333.563} C_DIS
LIN {X -0.006,Y -189.220,Z 1055.834,A 0.000,B 0.000,C 90.000,E1 330.205} C_DIS
LIN {X -0.043,Y -195.740,Z 1055.816,A 0.000,B 0.000,C 90.000,E1 326.914} C_DIS
LIN {X 0.085,Y -203.007,Z 1055.798,A 0.000,B 0.000,C 90.000,E1 323.623} C_DIS
LIN {X -0.066,Y -212.041,Z 1055.778,A 0.000,B 0.000,C 90.000,E1 320.070} C_DIS
LIN {X -0.030,Y -221.839,Z 1055.759,A 0.000,B 0.000,C 90.000,E1 316.539} C_DIS
LIN {X 0.018,Y -231.440,Z 1055.741,A 0.000,B 0.000,C 90.000,E1 313.461} C_DIS
LIN {X 0.034,Y -240.854,Z 1055.727,A 0.000,B 0.000,C 90.000,E1 310.825} C_DIS
LIN {X -0.034,Y -248.395,Z 1055.717,A 0.000,B 0.000,C 90.000,E1 308.991} C_DIS
LIN {X 0.027,Y -256.898,Z 1055.706,A 0.000,B 0.000,C 90.000,E1 307.156} C_DIS
LIN {X 0.023,Y -270.082,Z 1055.693,A 0.000,B 0.000,C 90.000,E1 304.659} C_DIS
LIN {X 0.046,Y -286.361,Z 1055.677,A 0.000,B 0.000,C 90.000,E1 301.878} C_DIS
LIN {X -0.036,Y -305.902,Z 1055.660,A 0.000,B 0.000,C 90.000,E1 298.871} C_DIS
LIN {X -0.096,Y -324.761,Z 1055.646,A 0.000,B 0.000,C 90.000,E1 296.283} C_DIS
LIN {X 0.000,Y -334.807,Z 1055.639,A 0.000,B 0.000,C 90.000,E1 295.027} C_DIS
LIN {X -0.013,Y -347.871,Z 1055.631,A 0.000,B 0.000,C 90.000,E1 293.590} C_DIS
LIN {X 0.019,Y -372.306,Z 1055.618,A 0.000,B 0.000,C 90.000,E1 291.227} C_DIS
LIN {X 0.035,Y -391.582,Z 1055.609,A 0.000,B 0.000,C 90.000,E1 289.523} C_DIS
LIN {X -0.021,Y -405.130,Z 1055.602,A 0.000,B 0.000,C 90.000,E1 288.362} C_DIS
LIN {X 0.085,Y -415.695,Z 1055.597,A 0.000,B 0.000,C 90.000,E1 287.402} C_DIS
LIN {X 0.089,Y -423.374,Z 1055.593,A 0.000,B 0.000,C 90.000,E1 286.677} C_DIS
LIN {X 0.220,Y -430.932,Z 1055.589,A 0.000,B 0.000,C 90.000,E1 285.898} C_DIS
LIN {X -0.151,Y -440.748,Z 1055.583,A 0.000,B 0.000,C 90.000,E1 284.898} C_DIS
LIN {X 0.177,Y -447.723,Z 1055.578,A 0.000,B 0.000,C 90.000,E1 284.064} C_DIS
LIN {X 0.020,Y -454.144,Z 1055.574,A 0.000,B 0.000,C 90.000,E1 283.300} C_DIS
LIN {X -0.088,Y -459.972,Z 1055.570,A 0.000,B 0.000,C 90.000,E1 282.535} C_DIS
LIN {X 0.151,Y -466.797,Z 1055.564,A 0.000,B 0.000,C 90.000,E1 281.478} C_DIS
LIN {X 0.156,Y -471.125,Z 1055.560,A 0.000,B 0.000,C 90.000,E1 280.715} C_DIS
LIN {X 0.106,Y -474.800,Z 1055.555,A 0.000,B 0.000,C 90.000,E1 279.962} C_DIS
LIN {X -0.246,Y -476.915,Z 1055.553,A 0.000,B 0.000,C 90.000,E1 279.500} C_DIS
LIN {X -0.037,Y -478.790,Z 1055.550,A 0.000,B 0.000,C 90.000,E1 278.973} C_DIS
LIN {X 0.104,Y -480.480,Z 1055.547,A 0.000,B 0.000,C 90.000,E1 278.454} C_DIS
LIN {X -0.218,Y -481.979,Z 1055.544,A 0.000,B 0.000,C 90.000,E1 277.992} C_DIS
LIN {X 0.011,Y -483.297,Z 1055.542,A 0.000,B 0.000,C 90.000,E1 277.466} C_DIS
LIN {X 0.184,Y -484.381,Z 1055.539,A 0.000,B 0.000,C 90.000,E1 276.947} C_DIS
LIN {X -0.116,Y -485.221,Z 1055.536,A 0.000,B 0.000,C 90.000,E1 276.486} C_DIS
LIN {X 0.071,Y -485.774,Z 1055.533,A 0.000,B 0.000,C 90.000,E1 275.967} C_DIS
LIN {X 0.217,Y -485.967,Z 1055.530,A 0.000,B 0.000,C 90.000,E1 275.454} C_DIS
LIN {X -0.069,Y -485.696,Z 1055.528,A 0.000,B 0.000,C 90.000,E1 274.992} C_DIS
LIN {X 0.129,Y -485.021,Z 1055.525,A 0.000,B 0.000,C 90.000,E1 274.473} C_DIS
LIN {X -0.162,Y -483.788,Z 1055.522,A 0.000,B 0.000,C 90.000,E1 274.012} C_DIS
LIN {X -0.007,Y -481.978,Z 1055.519,A 0.000,B 0.000,C 90.000,E1 273.498} C_DIS
LIN {X 0.171,Y -479.547,Z 1055.517,A 0.000,B 0.000,C 90.000,E1 272.980} C_DIS
LIN {X -0.173,Y -476.251,Z 1055.514,A 0.000,B 0.000,C 90.000,E1 272.522} C_DIS
LIN {X 0.125,Y -474.352,Z 1055.512,A 0.000,B 0.000,C 90.000,E1 272.236} C_DIS
LIN {X -0.221,Y -469.764,Z 1055.510,A 0.000,B 0.000,C 90.000,E1 271.776} C_DIS
LIN {X -0.003,Y -464.293,Z 1055.507,A 0.000,B 0.000,C 90.000,E1 271.260} C_DIS
LIN {X 0.035,Y -458.401,Z 1055.505,A 0.000,B 0.000,C 90.000,E1 270.802} C_DIS
LIN {X -0.010,Y -452.118,Z 1055.502,A 0.000,B 0.000,C 90.000,E1 270.401} C_DIS
LIN {X -0.063,Y -445.232,Z 1055.500,A 0.000,B 0.000,C 90.000,E1 270.057} C_DIS
LIN {X 0.025,Y -441.577,Z 1055.499,A 0.000,B 0.000,C 90.000,E1 269.885} C_DIS
LIN {X -0.115,Y -437.941,Z 1055.499,A 0.000,B 0.000,C 90.000,E1 269.771} C_DIS
LIN {X -0.095,Y -429.713,Z 1055.497,A 0.000,B 0.000,C 90.000,E1 269.542} C_DIS
LIN {X -0.005,Y -421.256,Z 1055.496,A 0.000,B 0.000,C 90.000,E1 269.370} C_DIS
LIN {X -0.004,Y -412.143,Z 1055.496,A 0.000,B 0.000,C 90.000,E1 269.255} C_DIS
LIN {X -0.190,Y -399.845,Z 1055.495,A 0.000,B 0.000,C 90.000,E1 269.198} C_DIS
LIN {X 0.083,Y -394.286,Z 1055.495,A 0.000,B 0.000,C 90.000,E1 269.141} C_DIS
LIN {X 0.010,Y -181.351,Z 1055.495,A 0.000,B 0.000,C 90.000,E1 269.141} C_DIS
LIN {X 0.067,Y -180.906,Z 1055.475,A 0.000,B 0.000,C 90.000,E1 265.412} C_DIS
LIN {X -0.057,Y -180.720,Z 1055.470,A 0.000,B 0.000,C 90.000,E1 264.609} C_DIS
LIN {X 0.041,Y -178.808,Z 1055.442,A 0.000,B 0.000,C 90.000,E1 259.511} C_DIS
LIN {X -0.052,Y -175.853,Z 1055.413,A 0.000,B 0.000,C 90.000,E1 254.448} C_DIS
LIN {X -0.070,Y -173.180,Z 1055.395,A 0.000,B 0.000,C 90.000,E1 251.040} C_DIS
LIN {X -0.067,Y -171.481,Z 1055.380,A 0.000,B 0.000,C 90.000,E1 248.465} C_DIS
LIN {X -0.080,Y -167.710,Z 1055.356,A 0.000,B 0.000,C 90.000,E1 244.152} C_DIS
LIN {X -0.063,Y -166.399,Z 1055.347,A 0.000,B 0.000,C 90.000,E1 242.410} C_DIS
LIN {X 0.076,Y -163.124,Z 1055.327,A 0.000,B 0.000,C 90.000,E1 238.869} C_DIS
LIN {X -0.098,Y -161.076,Z 1055.313,A 0.000,B 0.000,C 90.000,E1 236.294} C_DIS
LIN {X 0.012,Y -157.807,Z 1055.293,A 0.000,B 0.000,C 90.000,E1 232.718} C_DIS
LIN {X -0.050,Y -155.842,Z 1055.278,A 0.000,B 0.000,C 90.000,E1 230.070} C_DIS
LIN {X 0.007,Y -152.093,Z 1055.253,A 0.000,B 0.000,C 90.000,E1 225.567} C_DIS
LIN {X 0.026,Y -150.343,Z 1055.238,A 0.000,B 0.000,C 90.000,E1 222.852} C_DIS
LIN {X 0.046,Y -147.081,Z 1055.213,A 0.000,B 0.000,C 90.000,E1 218.302} C_DIS
LIN {X -0.050,Y -145.654,Z 1055.198,A 0.000,B 0.000,C 90.000,E1 215.598} C_DIS
LIN {X -0.046,Y -143.036,Z 1055.172,A 0.000,B 0.000,C 90.000,E1 211.003} C_DIS
LIN {X 0.081,Y -141.661,Z 1055.152,A 0.000,B 0.000,C 90.000,E1 207.257} C_DIS
LIN {X -0.001,Y -139.448,Z 1055.115,A 0.000,B 0.000,C 90.000,E1 200.791} C_DIS
LIN {X 0.052,Y -139.181,Z 1055.105,A 0.000,B 0.000,C 90.000,E1 198.906} C_DIS
LIN {X -0.056,Y -138.321,Z 1055.053,A 0.000,B 0.000,C 90.000,E1 189.613} C_DIS
LIN {X -0.049,Y -139.464,Z 1055.007,A 0.000,B 0.000,C 90.000,E1 181.203} C_DIS
LIN {X 0.030,Y -141.025,Z 1054.976,A 0.000,B 0.000,C 90.000,E1 175.584} C_DIS
LIN {X -0.014,Y -142.391,Z 1054.960,A 0.000,B 0.000,C 90.000,E1 172.818} C_DIS
LIN {X 0.048,Y -144.622,Z 1054.934,A 0.000,B 0.000,C 90.000,E1 168.173} C_DIS
LIN {X -0.033,Y -147.818,Z 1054.909,A 0.000,B 0.000,C 90.000,E1 163.614} C_DIS
LIN {X 0.053,Y -150.507,Z 1054.889,A 0.000,B 0.000,C 90.000,E1 159.934} C_DIS
LIN {X -0.066,Y -153.967,Z 1054.869,A 0.000,B 0.000,C 90.000,E1 156.357} C_DIS
LIN {X -0.004,Y -157.379,Z 1054.849,A 0.000,B 0.000,C 90.000,E1 152.743} C_DIS
LIN {X -0.063,Y -161.581,Z 1054.829,A 0.000,B 0.000,C 90.000,E1 149.203} C_DIS
LIN {X -0.051,Y -165.777,Z 1054.809,A 0.000,B 0.000,C 90.000,E1 145.674} C_DIS
LIN {X -0.065,Y -170.738,Z 1054.790,A 0.000,B 0.000,C 90.000,E1 142.190} C_DIS
LIN {X 0.093,Y -175.610,Z 1054.771,A 0.000,B 0.000,C 90.000,E1 138.690} C_DIS
LIN {X -0.037,Y -181.227,Z 1054.752,A 0.000,B 0.000,C 90.000,E1 135.324} C_DIS
LIN {X 0.094,Y -186.694,Z 1054.733,A 0.000,B 0.000,C 90.000,E1 131.919} C_DIS
LIN {X 0.046,Y -191.295,Z 1054.719,A 0.000,B 0.000,C 90.000,E1 129.439} C_DIS
LIN {X -0.003,Y -197.511,Z 1054.700,A 0.000,B 0.000,C 90.000,E1 125.964} C_DIS
LIN {X -0.032,Y -198.250,Z 1054.698,A 0.000,B 0.000,C 90.000,E1 125.598} C_DIS
LIN {X -0.091,Y -304.823,Z 1054.698,A 0.000,B 0.000,C 90.000,E1 125.598} C_DIS
LIN {X -0.050,Y -310.673,Z 1054.696,A 0.000,B 0.000,C 90.000,E1 125.358} C_DIS
LIN {X -0.107,Y -313.716,Z 1054.695,A 0.000,B 0.000,C 90.000,E1 125.105} C_DIS
LIN {X -0.153,Y -317.424,Z 1054.692,A 0.000,B 0.000,C 90.000,E1 124.612} C_DIS
LIN {X -0.095,Y -319.099,Z 1054.690,A 0.000,B 0.000,C 90.000,E1 124.278} C_DIS
LIN {X -0.045,Y -321.491,Z 1054.687,A 0.000,B 0.000,C 90.000,E1 123.627} C_DIS
LIN {X -0.182,Y -331.740,Z 1054.671,A 0.000,B 0.000,C 90.000,E1 120.797} C_DIS
LIN {X -0.063,Y -343.320,Z 1054.655,A 0.000,B 0.000,C 90.000,E1 117.975} C_DIS
LIN {X 0.067,Y -356.339,Z 1054.640,A 0.000,B 0.000,C 90.000,E1 115.207} C_DIS
LIN {X 0.034,Y -369.208,Z 1054.627,A 0.000,B 0.000,C 90.000,E1 112.823} C_DIS
LIN {X 0.036,Y -383.394,Z 1054.614,A 0.000,B 0.000,C 90.000,E1 110.482} C_DIS
LIN {X 0.136,Y -398.995,Z 1054.601,A 0.000,B 0.000,C 90.000,E1 108.181} C_DIS
LIN {X 0.002,Y -416.124,Z 1054.589,A 0.000,B 0.000,C 90.000,E1 105.969} C_DIS
LIN {X 0.181,Y -434.902,Z 1054.577,A 0.000,B 0.000,C 90.000,E1 103.772} C_DIS
LIN {X 0.195,Y -454.884,Z 1054.565,A 0.000,B 0.000,C 90.000,E1 101.715} C_DIS
LIN {X -0.033,Y -467.610,Z 1054.559,A 0.000,B 0.000,C 90.000,E1 100.546} C_DIS
LIN {X -0.014,Y -469.631,Z 1054.557,A 0.000,B 0.000,C 90.000,E1 100.310} C_DIS
LIN {X -0.165,Y -471.289,Z 1054.556,A 0.000,B 0.000,C 90.000,E1 100.074} C_DIS
LIN {X 0.067,Y -472.532,Z 1054.554,A 0.000,B 0.000,C 90.000,E1 99.792} C_DIS
LIN {X -0.217,Y -474.061,Z 1054.552,A 0.000,B 0.000,C 90.000,E1 99.321} C_DIS
LIN {X -0.104,Y -474.547,Z 1054.549,A 0.000,B 0.000,C 90.000,E1 98.803} C_DIS
LIN {X 0.090,Y -474.069,Z 1054.546,A 0.000,B 0.000,C 90.000,E1 98.276} C_DIS
LIN {X 0.215,Y -472.558,Z 1054.543,A 0.000,B 0.000,C 90.000,E1 97.757} C_DIS
LIN {X 0.013,Y -471.337,Z 1054.542,A 0.000,B 0.000,C 90.000,E1 97.530} C_DIS
LIN {X -0.017,Y -466.130,Z 1054.538,A 0.000,B 0.000,C 90.000,E1 96.777} C_DIS
LIN {X 0.185,Y -455.468,Z 1054.529,A 0.000,B 0.000,C 90.000,E1 95.220} C_DIS
LIN {X -0.149,Y -439.553,Z 1054.516,A 0.000,B 0.000,C 90.000,E1 92.922} C_DIS
LIN {X 0.029,Y -418.929,Z 1054.497,A 0.000,B 0.000,C 90.000,E1 89.427} C_DIS
LIN {X -0.049,Y -407.210,Z 1054.485,A 0.000,B 0.000,C 90.000,E1 87.249} C_DIS
LIN {X -0.059,Y -398.240,Z 1054.475,A 0.000,B 0.000,C 90.000,E1 85.584} C_DIS
LIN {X 0.198,Y -389.075,Z 1054.466,A 0.000,B 0.000,C 90.000,E1 83.856} C_DIS
LIN {X -0.079,Y -378.177,Z 1054.455,A 0.000,B 0.000,C 90.000,E1 81.894} C_DIS
LIN {X -0.086,Y -368.476,Z 1054.445,A 0.000,B 0.000,C 90.000,E1 80.151} C_DIS
LIN {X 0.121,Y -356.790,Z 1054.434,A 0.000,B 0.000,C 90.000,E1 78.049} C_DIS
LIN {X 0.139,Y -345.166,Z 1054.422,A 0.000,B 0.000,C 90.000,E1 75.936} C_DIS
LIN {X -0.054,Y -330.597,Z 1054.407,A 0.000,B 0.000,C 90.000,E1 73.196} C_DIS
LIN {X -0.132,Y -316.583,Z 1054.391,A 0.000,B 0.000,C 90.000,E1 70.369} C_DIS
LIN {X -0.173,Y -304.648,Z 1054.376,A 0.000,B 0.000,C 90.000,E1 67.794} C_DIS
LIN {X 0.115,Y -293.121,Z 1054.362,A 0.000,B 0.000,C 90.000,E1 65.101} C_DIS
LIN {X 0.130,Y -283.240,Z 1054.349,A 0.000,B 0.000,C 90.000,E1 62.743} C_DIS
LIN {X 0.125,Y -272.169,Z 1054.333,A 0.000,B 0.000,C 90.000,E1 59.999} C_DIS
LIN {X -0.021,Y -262.678,Z 1054.320,A 0.000,B 0.000,C 90.000,E1 57.582} C_DIS
LIN {X 0.035,Y -250.851,Z 1054.302,A 0.000,B 0.000,C 90.000,E1 54.356} C_DIS
LIN {X -0.051,Y -240.766,Z 1054.286,A 0.000,B 0.000,C 90.000,E1 51.457} C_DIS
LIN {X 0.034,Y -230.112,Z 1054.267,A 0.000,B 0.000,C 90.000,E1 48.081} C_DIS
LIN {X -0.045,Y -220.306,Z 1054.248,A 0.000,B 0.000,C 90.000,E1 44.676} C_DIS
LIN {X 0.048,Y -212.086,Z 1054.231,A 0.000,B 0.000,C 90.000,E1 41.553} C_DIS
LIN {X 0.108,Y -204.327,Z 1054.213,A 0.000,B 0.000,C 90.000,E1 38.382} C_DIS
LIN {X -0.085,Y -197.125,Z 1054.196,A 0.000,B 0.000,C 90.000,E1 35.231} C_DIS
LIN {X 0.079,Y -190.578,Z 1054.177,A 0.000,B 0.000,C 90.000,E1 31.926} C_DIS
LIN {X 0.101,Y -184.723,Z 1054.159,A 0.000,B 0.000,C 90.000,E1 28.615} C_DIS
LIN {X 0.048,Y -179.593,Z 1054.141,A 0.000,B 0.000,C 90.000,E1 25.283} C_DIS
LIN {X 0.046,Y -175.237,Z 1054.122,A 0.000,B 0.000,C 90.000,E1 21.897} C_DIS
LIN {X 0.009,Y -171.577,Z 1054.103,A 0.000,B 0.000,C 90.000,E1 18.489} C_DIS
LIN {X 0.006,Y -167.947,Z 1054.079,A 0.000,B 0.000,C 90.000,E1 14.175} C_DIS
LIN {X -0.062,Y -165.447,Z 1054.055,A 0.000,B 0.000,C 90.000,E1 9.849} C_DIS
LIN {X 0.039,Y -163.454,Z 1054.016,A 0.000,B 0.000,C 90.000,E1 2.808} C_DIS
LIN {X -0.022,Y -164.745,Z 1053.963,A 0.000,B 0.000,C 90.000,E1 353.394} C_DIS
LIN {X 0.069,Y -167.412,Z 1053.934,A 0.000,B 0.000,C 90.000,E1 348.117} C_DIS
LIN {X 0.008,Y -170.779,Z 1053.910,A 0.000,B 0.000,C 90.000,E1 343.795} C_DIS
LIN {X -0.062,Y -174.248,Z 1053.891,A 0.000,B 0.000,C 90.000,E1 340.369} C_DIS
LIN {X 0.022,Y -178.450,Z 1053.872,A 0.000,B 0.000,C 90.000,E1 336.922} C_DIS
LIN {X 0.098,Y -183.384,Z 1053.853,A 0.000,B 0.000,C 90.000,E1 333.512} C_DIS
LIN {X -0.034,Y -189.133,Z 1053.834,A 0.000,B 0.000,C 90.000,E1 330.205} C_DIS
LIN {X -0.074,Y -195.661,Z 1053.816,A 0.000,B 0.000,C 90.000,E1 326.914} C_DIS
LIN {X 0.050,Y -202.946,Z 1053.798,A 0.000,B 0.000,C 90.000,E1 323.623} C_DIS
LIN {X -0.098,Y -211.956,Z 1053.778,A 0.000,B 0.000,C 90.000,E1 320.070} C_DIS
LIN {X -0.066,Y -221.736,Z 1053.758,A 0.000,B 0.000,C 90.000,E1 316.539} C_DIS
LIN {X -0.022,Y -231.345,Z 1053.741,A 0.000,B 0.000,C 90.000,E1 313.461} C_DIS
LIN {X -0.010,Y -240.732,Z 1053.727,A 0.000,B 0.000,C 90.000,E1 310.825} C_DIS
LIN {X -0.081,Y -248.268,Z 1053.717,A 0.000,B 0.000,C 90.000,E1 308.991} C_DIS
LIN {X -0.047,Y -254.996,Z 1053.708,A 0.000,B 0.000,C 90.000,E1 307.523} C_DIS
LIN {X -0.089,Y -268.051,Z 1053.694,A 0.000,B 0.000,C 90.000,E1 305.025} C_DIS
LIN {X -0.015,Y -286.299,Z 1053.677,A 0.000,B 0.000,C 90.000,E1 301.878} C_DIS
LIN {X -0.103,Y -305.889,Z 1053.660,A 0.000,B 0.000,C 90.000,E1 298.871} C_DIS
LIN {X 0.125,Y -324.811,Z 1053.646,A 0.000,B 0.000,C 90.000,E1 296.232} C_DIS
LIN {X 0.018,Y -337.463,Z 1053.637,A 0.000,B 0.000,C 90.000,E1 294.719} C_DIS
LIN {X 0.127,Y -350.967,Z 1053.629,A 0.000,B 0.000,C 90.000,E1 293.259} C_DIS
LIN {X -0.170,Y -372.736,Z 1053.618,A 0.000,B 0.000,C 90.000,E1 291.227} C_DIS
LIN {X -0.038,Y -392.066,Z 1053.608,A 0.000,B 0.000,C 90.000,E1 289.504} C_DIS
LIN {X 0.131,Y -405.597,Z 1053.602,A 0.000,B 0.000,C 90.000,E1 288.308} C_DIS
LIN {X -0.188,Y -416.197,Z 1053.597,A 0.000,B 0.000,C 90.000,E1 287.402} C_DIS
LIN {X 0.186,Y -423.857,Z 1053.593,A 0.000,B 0.000,C 90.000,E1 286.622} C_DIS
LIN {X -0.130,Y -431.410,Z 1053.588,A 0.000,B 0.000,C 90.000,E1 285.898} C_DIS
LIN {X 0.222,Y -438.779,Z 1053.584,A 0.000,B 0.000,C 90.000,E1 285.064} C_DIS
LIN {X -0.228,Y -448.167,Z 1053.578,A 0.000,B 0.000,C 90.000,E1 284.064} C_DIS
LIN {X -0.135,Y -456.554,Z 1053.572,A 0.000,B 0.000,C 90.000,E1 283.008} C_DIS
LIN {X -0.217,Y -462.092,Z 1053.568,A 0.000,B 0.000,C 90.000,E1 282.243} C_DIS
LIN {X 0.199,Y -467.075,Z 1053.564,A 0.000,B 0.000,C 90.000,E1 281.422} C_DIS
LIN {X 0.207,Y -471.408,Z 1053.559,A 0.000,B 0.000,C 90.000,E1 280.658} C_DIS
LIN {X 0.161,Y -475.072,Z 1053.555,A 0.000,B 0.000,C 90.000,E1 279.905} C_DIS
LIN {X -0.110,Y -477.177,Z 1053.552,A 0.000,B 0.000,C 90.000,E1 279.434} C_DIS
LIN {X 0.023,Y -479.051,Z 1053.550,A 0.000,B 0.000,C 90.000,E1 278.916} C_DIS
LIN {X 0.166,Y -480.737,Z 1053.547,A 0.000,B 0.000,C 90.000,E1 278.398} C_DIS
LIN {X -0.153,Y -482.227,Z 1053.544,A 0.000,B 0.000,C 90.000,E1 277.936} C_DIS
LIN {X 0.077,Y -483.523,Z 1053.541,A 0.000,B 0.000,C 90.000,E1 277.409} C_DIS
LIN {X 0.253,Y -484.601,Z 1053.538,A 0.000,B 0.000,C 90.000,E1 276.891} C_DIS
LIN {X -0.045,Y -485.418,Z 1053.536,A 0.000,B 0.000,C 90.000,E1 276.429} C_DIS
LIN {X 0.144,Y -485.948,Z 1053.533,A 0.000,B 0.000,C 90.000,E1 275.910} C_DIS
LIN {X -0.146,Y -486.111,Z 1053.530,A 0.000,B 0.000,C 90.000,E1 275.448} C_DIS
LIN {X 0.007,Y -485.850,Z 1053.527,A 0.000,B 0.000,C 90.000,E1 274.935} C_DIS
LIN {X 0.205,Y -485.080,Z 1053.525,A 0.000,B 0.000,C 90.000,E1 274.416} C_DIS
LIN {X -0.085,Y -483.806,Z 1053.522,A 0.000,B 0.000,C 90.000,E1 273.955} C_DIS
LIN {X 0.071,Y -481.939,Z 1053.519,A 0.000,B 0.000,C 90.000,E1 273.440} C_DIS
LIN {X -0.231,Y -479.434,Z 1053.516,A 0.000,B 0.000,C 90.000,E1 272.980} C_DIS
LIN {X -0.096,Y -476.147,Z 1053.514,A 0.000,B 0.000,C 90.000,E1 272.465} C_DIS
LIN {X 0.024,Y -471.938,Z 1053.511,A 0.000,B 0.000,C 90.000,E1 271.949} C_DIS
LIN {X 0.136,Y -466.715,Z 1053.508,A 0.000,B 0.000,C 90.000,E1 271.432} C_DIS
LIN {X 0.027,Y -461.003,Z 1053.505,A 0.000,B 0.000,C 90.000,E1 270.974} C_DIS
LIN {X -0.204,Y -454.818,Z 1053.503,A 0.000,B 0.000,C 90.000,E1 270.573} C_DIS
LIN {X 0.117,Y -451.739,Z 1053.502,A 0.000,B 0.000,C 90.000,E1 270.344} C_DIS
LIN {X 0.096,Y -444.871,Z 1053.500,A 0.000,B 0.000,C 90.000,E1 270.000} C_DIS
LIN {X 0.207,Y -441.192,Z 1053.499,A 0.000,B 0.000,C 90.000,E1 269.828} C_DIS
LIN {X -0.028,Y -433.092,Z 1053.498,A 0.000,B 0.000,C 90.000,E1 269.599} C_DIS
LIN {X -0.112,Y -424.822,Z 1053.497,A 0.000,B 0.000,C 90.000,E1 269.427} C_DIS
LIN {X 0.204,Y -416.020,Z 1053.496,A 0.000,B 0.000,C 90.000,E1 269.255} C_DIS
LIN {X -0.180,Y -402.838,Z 1053.495,A 0.000,B 0.000,C 90.000,E1 269.198} C_DIS
LIN {X -0.024,Y -389.841,Z 1053.495,A 0.000,B 0.000,C 90.000,E1 269.141} C_DIS
LIN {X -0.039,Y -181.348,Z 1053.495,A 0.000,B 0.000,C 90.000,E1 269.141} C_DIS
LIN {X 0.018,Y -180.906,Z 1053.474,A 0.000,B 0.000,C 90.000,E1 265.412} C_DIS
LIN {X 0.075,Y -180.712,Z 1053.470,A 0.000,B 0.000,C 90.000,E1 264.552} C_DIS
LIN {X -0.007,Y -178.799,Z 1053.442,A 0.000,B 0.000,C 90.000,E1 259.511} C_DIS
LIN {X 0.070,Y -175.845,Z 1053.413,A 0.000,B 0.000,C 90.000,E1 254.393} C_DIS
LIN {X 0.069,Y -172.036,Z 1053.385,A 0.000,B 0.000,C 90.000,E1 249.263} C_DIS
LIN {X 0.046,Y -171.467,Z 1053.380,A 0.000,B 0.000,C 90.000,E1 248.411} C_DIS
LIN {X 0.025,Y -167.699,Z 1053.356,A 0.000,B 0.000,C 90.000,E1 244.101} C_DIS
LIN {X 0.039,Y -166.383,Z 1053.347,A 0.000,B 0.000,C 90.000,E1 242.359} C_DIS
LIN {X 0.031,Y -163.111,Z 1053.327,A 0.000,B 0.000,C 90.000,E1 238.869} C_DIS
LIN {X 0.080,Y -161.059,Z 1053.313,A 0.000,B 0.000,C 90.000,E1 236.215} C_DIS
LIN {X -0.032,Y -157.794,Z 1053.293,A 0.000,B 0.000,C 90.000,E1 232.718} C_DIS
LIN {X 0.007,Y -155.830,Z 1053.278,A 0.000,B 0.000,C 90.000,E1 230.033} C_DIS
LIN {X -0.037,Y -152.081,Z 1053.253,A 0.000,B 0.000,C 90.000,E1 225.567} C_DIS
LIN {X -0.018,Y -150.331,Z 1053.238,A 0.000,B 0.000,C 90.000,E1 222.852} C_DIS
LIN {X 0.004,Y -147.072,Z 1053.213,A 0.000,B 0.000,C 90.000,E1 218.302} C_DIS
LIN {X -0.092,Y -145.646,Z 1053.198,A 0.000,B 0.000,C 90.000,E1 215.598} C_DIS
LIN {X -0.088,Y -143.029,Z 1053.172,A 0.000,B 0.000,C 90.000,E1 211.003} C_DIS
LIN {X 0.039,Y -141.654,Z 1053.151,A 0.000,B 0.000,C 90.000,E1 207.257} C_DIS
LIN {X -0.041,Y -139.445,Z 1053.115,A 0.000,B 0.000,C 90.000,E1 200.791} C_DIS
LIN {X 0.010,Y -139.178,Z 1053.105,A 0.000,B 0.000,C 90.000,E1 198.906} C_DIS
LIN {X 0.039,Y -138.320,Z 1053.053,A 0.000,B 0.000,C 90.000,E1 189.557} C_DIS
LIN {X 0.048,Y -139.467,Z 1053.006,A 0.000,B 0.000,C 90.000,E1 181.146} C_DIS
LIN {X -0.011,Y -141.033,Z 1052.975,A 0.000,B 0.000,C 90.000,E1 175.584} C_DIS
LIN {X -0.057,Y -142.400,Z 1052.960,A 0.000,B 0.000,C 90.000,E1 172.818} C_DIS
LIN {X 0.006,Y -144.632,Z 1052.934,A 0.000,B 0.000,C 90.000,E1 168.173} C_DIS
LIN {X 0.066,Y -147.828,Z 1052.909,A 0.000,B 0.000,C 90.000,E1 163.559} C_DIS
LIN {X 0.010,Y -150.521,Z 1052.889,A 0.000,B 0.000,C 90.000,E1 159.934} C_DIS
LIN {X 0.030,Y -153.983,Z 1052.868,A 0.000,B 0.000,C 90.000,E1 156.305} C_DIS
LIN {X -0.049,Y -157.396,Z 1052.849,A 0.000,B 0.000,C 90.000,E1 152.743} C_DIS
LIN {X 0.032,Y -161.601,Z 1052.829,A 0.000,B 0.000,C 90.000,E1 149.154} C_DIS
LIN {X -0.097,Y -165.798,Z 1052.809,A 0.000,B 0.000,C 90.000,E1 145.674} C_DIS
LIN {X 0.022,Y -170.762,Z 1052.790,A 0.000,B 0.000,C 90.000,E1 142.145} C_DIS
LIN {X 0.045,Y -175.634,Z 1052.771,A 0.000,B 0.000,C 90.000,E1 138.690} C_DIS
LIN {X -0.086,Y -181.249,Z 1052.752,A 0.000,B 0.000,C 90.000,E1 135.324} C_DIS
LIN {X 0.045,Y -186.721,Z 1052.733,A 0.000,B 0.000,C 90.000,E1 131.919} C_DIS
LIN {X -0.005,Y -191.319,Z 1052.719,A 0.000,B 0.000,C 90.000,E1 129.439} C_DIS
LIN {X 0.065,Y -197.539,Z 1052.700,A 0.000,B 0.000,C 90.000,E1 125.931} C_DIS
LIN {X -0.028,Y -198.155,Z 1052.698,A 0.000,B 0.000,C 90.000,E1 125.644} C_DIS
LIN {X 0.151,Y -304.176,Z 1052.698,A 0.000,B 0.000,C 90.000,E1 125.598} C_DIS
LIN {X 0.049,Y -309.040,Z 1052.697,A 0.000,B 0.000,C 90.000,E1 125.471} C_DIS
LIN {X 0.123,Y -311.282,Z 1052.696,A 0.000,B 0.000,C 90.000,E1 125.311} C_DIS
LIN {X -0.025,Y -315.150,Z 1052.694,A 0.000,B 0.000,C 90.000,E1 124.945} C_DIS
LIN {X -0.185,Y -318.618,Z 1052.691,A 0.000,B 0.000,C 90.000,E1 124.405} C_DIS
LIN {X 0.057,Y -319.998,Z 1052.689,A 0.000,B 0.000,C 90.000,E1 124.040} C_DIS
LIN {X 0.102,Y -332.518,Z 1052.670,A 0.000,B 0.000,C 90.000,E1 120.541} C_DIS
LIN {X -0.047,Y -344.199,Z 1052.654,A 0.000,B 0.000,C 90.000,E1 117.769} C_DIS
LIN {X -0.048,Y -357.328,Z 1052.639,A 0.000,B 0.000,C 90.000,E1 115.027} C_DIS
LIN {X -0.057,Y -370.302,Z 1052.626,A 0.000,B 0.000,C 90.000,E1 112.642} C_DIS
LIN {X -0.026,Y -384.599,Z 1052.613,A 0.000,B 0.000,C 90.000,E1 110.301} C_DIS
LIN {X 0.103,Y -400.321,Z 1052.600,A 0.000,B 0.000,C 90.000,E1 108.000} C_DIS
LIN {X 0.000,Y -417.580,Z 1052.588,A 0.000,B 0.000,C 90.000,E1 105.788} C_DIS
LIN {X 0.212,Y -436.501,Z 1052.576,A 0.000,B 0.000,C 90.000,E1 103.592} C_DIS
LIN {X -0.109,Y -456.532,Z 1052.564,A 0.000,B 0.000,C 90.000,E1 101.591} C_DIS
LIN {X 0.144,Y -466.758,Z 1052.559,A 0.000,B 0.000,C 90.000,E1 100.602} C_DIS
LIN {X 0.178,Y -468.978,Z 1052.558,A 0.000,B 0.000,C 90.000,E1 100.366} C_DIS
LIN {X 0.127,Y -470.655,Z 1052.556,A 0.000,B 0.000,C 90.000,E1 100.141} C_DIS
LIN {X -0.020,Y -472.051,Z 1052.555,A 0.000,B 0.000,C 90.000,E1 99.905} C_DIS
LIN {X -0.168,Y -473.089,Z 1052.554,A 0.000,B 0.000,C 90.000,E1 99.670} C_DIS
LIN {X -0.060,Y -474.290,Z 1052.551,A 0.000,B 0.000,C 90.000,E1 99.151} C_DIS
LIN {X 0.131,Y -474.488,Z 1052.548,A 0.000,B 0.000,C 90.000,E1 98.624} C_DIS
LIN {X -0.213,Y -473.720,Z 1052.545,A 0.000,B 0.000,C 90.000,E1 98.163} C_DIS
LIN {X -0.086,Y -471.862,Z 1052.542,A 0.000,B 0.000,C 90.000,E1 97.644} C_DIS
LIN {X 0.240,Y -470.413,Z 1052.541,A 0.000,B 0.000,C 90.000,E1 97.352} C_DIS
LIN {X -0.168,Y -457.979,Z 1052.531,A 0.000,B 0.000,C 90.000,E1 95.625} C_DIS
LIN {X -0.034,Y -438.548,Z 1052.515,A 0.000,B 0.000,C 90.000,E1 92.751} C_DIS
LIN {X 0.103,Y -418.032,Z 1052.496,A 0.000,B 0.000,C 90.000,E1 89.255} C_DIS
LIN {X 0.001,Y -406.334,Z 1052.484,A 0.000,B 0.000,C 90.000,E1 87.078} C_DIS
LIN {X -0.028,Y -397.343,Z 1052.474,A 0.000,B 0.000,C 90.000,E1 85.412} C_DIS
LIN {X -0.177,Y -388.188,Z 1052.465,A 0.000,B 0.000,C 90.000,E1 83.742} C_DIS
LIN {X -0.057,Y -378.833,Z 1052.456,A 0.000,B 0.000,C 90.000,E1 82.008} C_DIS
LIN {X -0.111,Y -369.151,Z 1052.446,A 0.000,B 0.000,C 90.000,E1 80.274} C_DIS
LIN {X 0.136,Y -359.140,Z 1052.436,A 0.000,B 0.000,C 90.000,E1 78.465} C_DIS
LIN {X 0.130,Y -345.851,Z 1052.423,A 0.000,B 0.000,C 90.000,E1 76.061} C_DIS
LIN {X -0.057,Y -331.245,Z 1052.407,A 0.000,B 0.000,C 90.000,E1 73.323} C_DIS
LIN {X -0.012,Y -317.223,Z 1052.391,A 0.000,B 0.000,C 90.000,E1 70.477} C_DIS
LIN {X -0.032,Y -305.259,Z 1052.377,A 0.000,B 0.000,C 90.000,E1 67.901} C_DIS
LIN {X -0.115,Y -295.122,Z 1052.364,A 0.000,B 0.000,C 90.000,E1 65.613} C_DIS
LIN {X -0.079,Y -283.780,Z 1052.349,A 0.000,B 0.000,C 90.000,E1 62.922} C_DIS
LIN {X 0.181,Y -272.689,Z 1052.334,A 0.000,B 0.000,C 90.000,E1 60.127} C_DIS
LIN {X 0.050,Y -263.193,Z 1052.321,A 0.000,B 0.000,C 90.000,E1 57.709} C_DIS
LIN {X 0.117,Y -251.304,Z 1052.303,A 0.000,B 0.000,C 90.000,E1 54.482} C_DIS
LIN {X -0.101,Y -242.429,Z 1052.289,A 0.000,B 0.000,C 90.000,E1 51.984} C_DIS
LIN {X 0.030,Y -231.643,Z 1052.270,A 0.000,B 0.000,C 90.000,E1 48.609} C_DIS
LIN {X -0.009,Y -221.681,Z 1052.251,A 0.000,B 0.000,C 90.000,E1 45.202} C_DIS
LIN {X -0.049,Y -213.399,Z 1052.234,A 0.000,B 0.000,C 90.000,E1 42.123} C_DIS
LIN {X 0.041,Y -205.533,Z 1052.216,A 0.000,B 0.000,C 90.000,E1 38.955} C_DIS
LIN {X -0.122,Y -198.238,Z 1052.199,A 0.000,B 0.000,C 90.000,E1 35.804} C_DIS
LIN {X -0.087,Y -191.524,Z 1052.181,A 0.000,B 0.000,C 90.000,E1 32.546} C_DIS
LIN {X 0.058,Y -185.555,Z 1052.162,A 0.000,B 0.000,C 90.000,E1 29.205} C_DIS
LIN {X -0.055,Y -180.283,Z 1052.144,A 0.000,B 0.000,C 90.000,E1 25.899} C_DIS
LIN {X -0.042,Y -175.797,Z 1052.125,A 0.000,B 0.000,C 90.000,E1 22.514} C_DIS
LIN {X -0.007,Y -171.978,Z 1052.106,A 0.000,B 0.000,C 90.000,E1 19.087} C_DIS
LIN {X 0.003,Y -168.235,Z 1052.082,A 0.000,B 0.000,C 90.000,E1 14.773} C_DIS
LIN {X -0.019,Y -165.557,Z 1052.058,A 0.000,B 0.000,C 90.000,E1 10.433} C_DIS
LIN {X -0.052,Y -163.384,Z 1052.019,A 0.000,B 0.000,C 90.000,E1 3.440} C_DIS
LIN {X -0.027,Y -164.612,Z 1051.963,A 0.000,B 0.000,C 90.000,E1 353.394} C_DIS
LIN {X 0.058,Y -167.271,Z 1051.934,A 0.000,B 0.000,C 90.000,E1 348.117} C_DIS
LIN {X -0.006,Y -170.652,Z 1051.910,A 0.000,B 0.000,C 90.000,E1 343.795} C_DIS
LIN {X -0.080,Y -174.146,Z 1051.891,A 0.000,B 0.000,C 90.000,E1 340.369} C_DIS
LIN {X 0.001,Y -178.339,Z 1051.872,A 0.000,B 0.000,C 90.000,E1 336.922} C_DIS
LIN {X 0.074,Y -183.293,Z 1051.853,A 0.000,B 0.000,C 90.000,E1 333.512} C_DIS
LIN {X -0.061,Y -189.041,Z 1051.834,A 0.000,B 0.000,C 90.000,E1 330.205} C_DIS
LIN {X -0.105,Y -195.581,Z 1051.816,A 0.000,B 0.000,C 90.000,E1 326.914} C_DIS
LIN {X 0.017,Y -202.886,Z 1051.798,A 0.000,B 0.000,C 90.000,E1 323.623} C_DIS
LIN {X -0.036,Y -210.848,Z 1051.780,A 0.000,B 0.000,C 90.000,E1 320.436} C_DIS
LIN {X -0.026,Y -220.531,Z 1051.760,A 0.000,B 0.000,C 90.000,E1 316.905} C_DIS
LIN {X -0.004,Y -230.000,Z 1051.743,A 0.000,B 0.000,C 90.000,E1 313.824} C_DIS
LIN {X 0.142,Y -239.228,Z 1051.729,A 0.000,B 0.000,C 90.000,E1 311.148} C_DIS
LIN {X 0.024,Y -246.577,Z 1051.719,A 0.000,B 0.000,C 90.000,E1 309.322} C_DIS
LIN {X -0.121,Y -253.137,Z 1051.710,A 0.000,B 0.000,C 90.000,E1 307.890} C_DIS
LIN {X -0.058,Y -266.030,Z 1051.696,A 0.000,B 0.000,C 90.000,E1 305.358} C_DIS
LIN {X -0.042,Y -284.181,Z 1051.679,A 0.000,B 0.000,C 90.000,E1 302.212} C_DIS
LIN {X 0.065,Y -303.672,Z 1051.662,A 0.000,B 0.000,C 90.000,E1 299.155} C_DIS
LIN {X 0.046,Y -319.983,Z 1051.649,A 0.000,B 0.000,C 90.000,E1 296.873} C_DIS
LIN {X -0.090,Y -332.366,Z 1051.641,A 0.000,B 0.000,C 90.000,E1 295.335} C_DIS
LIN {X 0.010,Y -345.756,Z 1051.632,A 0.000,B 0.000,C 90.000,E1 293.823} C_DIS
LIN {X 0.179,Y -370.244,Z 1051.619,A 0.000,B 0.000,C 90.000,E1 291.408} C_DIS
LIN {X -0.216,Y -389.524,Z 1051.610,A 0.000,B 0.000,C 90.000,E1 289.758} C_DIS
LIN {X 0.051,Y -403.140,Z 1051.603,A 0.000,B 0.000,C 90.000,E1 288.544} C_DIS
LIN {X -0.129,Y -413.621,Z 1051.598,A 0.000,B 0.000,C 90.000,E1 287.638} C_DIS
LIN {X -0.176,Y -421.458,Z 1051.594,A 0.000,B 0.000,C 90.000,E1 286.913} C_DIS
LIN {X -0.020,Y -429.004,Z 1051.590,A 0.000,B 0.000,C 90.000,E1 286.134} C_DIS
LIN {X -0.153,Y -436.419,Z 1051.585,A 0.000,B 0.000,C 90.000,E1 285.371} C_DIS
LIN {X -0.033,Y -445.896,Z 1051.579,A 0.000,B 0.000,C 90.000,E1 284.300} C_DIS
LIN {X -0.215,Y -452.453,Z 1051.575,A 0.000,B 0.000,C 90.000,E1 283.536} C_DIS
LIN {X 0.112,Y -458.447,Z 1051.571,A 0.000,B 0.000,C 90.000,E1 282.715} C_DIS
LIN {X 0.044,Y -463.835,Z 1051.566,A 0.000,B 0.000,C 90.000,E1 281.951} C_DIS
LIN {X 0.025,Y -468.619,Z 1051.562,A 0.000,B 0.000,C 90.000,E1 281.186} C_DIS
LIN {X -0.047,Y -472.750,Z 1051.558,A 0.000,B 0.000,C 90.000,E1 280.433} C_DIS
LIN {X 0.006,Y -476.222,Z 1051.554,A 0.000,B 0.000,C 90.000,E1 279.670} C_DIS
LIN {X 0.003,Y -479.153,Z 1051.550,A 0.000,B 0.000,C 90.000,E1 278.916} C_DIS
LIN {X 0.146,Y -480.852,Z 1051.547,A 0.000,B 0.000,C 90.000,E1 278.398} C_DIS
LIN {X -0.173,Y -482.336,Z 1051.544,A 0.000,B 0.000,C 90.000,E1 277.936} C_DIS
LIN {X 0.059,Y -483.641,Z 1051.541,A 0.000,B 0.000,C 90.000,E1 277.409} C_DIS
LIN {X 0.235,Y -484.733,Z 1051.538,A 0.000,B 0.000,C 90.000,E1 276.891} C_DIS
LIN {X -0.063,Y -485.570,Z 1051.536,A 0.000,B 0.000,C 90.000,E1 276.429} C_DIS
LIN {X 0.127,Y -486.089,Z 1051.533,A 0.000,B 0.000,C 90.000,E1 275.910} C_DIS
LIN {X -0.162,Y -486.243,Z 1051.530,A 0.000,B 0.000,C 90.000,E1 275.448} C_DIS
LIN {X -0.008,Y -485.999,Z 1051.527,A 0.000,B 0.000,C 90.000,E1 274.935} C_DIS
LIN {X 0.191,Y -485.251,Z 1051.525,A 0.000,B 0.000,C 90.000,E1 274.416} C_DIS
LIN {X -0.098,Y -483.985,Z 1051.522,A 0.000,B 0.000,C 90.000,E1 273.955} C_DIS
LIN {X 0.059,Y -482.101,Z 1051.519,A 0.000,B 0.000,C 90.000,E1 273.440} C_DIS
LIN {X 0.236,Y -479.578,Z 1051.516,A 0.000,B 0.000,C 90.000,E1 272.922} C_DIS
LIN {X -0.106,Y -476.288,Z 1051.514,A 0.000,B 0.000,C 90.000,E1 272.465} C_DIS
LIN {X 0.016,Y -472.074,Z 1051.511,A 0.000,B 0.000,C 90.000,E1 271.949} C_DIS
LIN {X -0.155,Y -469.636,Z 1051.509,A 0.000,B 0.000,C 90.000,E1 271.718} C_DIS
LIN {X 0.092,Y -464.180,Z 1051.507,A 0.000,B 0.000,C 90.000,E1 271.203} C_DIS
LIN {X 0.186,Y -458.393,Z 1051.504,A 0.000,B 0.000,C 90.000,E1 270.745} C_DIS
LIN {X 0.169,Y -452.108,Z 1051.502,A 0.000,B 0.000,C 90.000,E1 270.344} C_DIS
LIN {X 0.107,Y -445.350,Z 1051.500,A 0.000,B 0.000,C 90.000,E1 270.000} C_DIS
LIN {X 0.185,Y -441.568,Z 1051.499,A 0.000,B 0.000,C 90.000,E1 269.828} C_DIS
LIN {X -0.049,Y -433.588,Z 1051.498,A 0.000,B 0.000,C 90.000,E1 269.599} C_DIS
LIN {X -0.162,Y -425.306,Z 1051.497,A 0.000,B 0.000,C 90.000,E1 269.427} C_DIS
LIN {X 0.124,Y -416.170,Z 1051.496,A 0.000,B 0.000,C 90.000,E1 269.255} C_DIS
LIN {X 0.154,Y -403.160,Z 1051.495,A 0.000,B 0.000,C 90.000,E1 269.141} C_DIS
LIN {X -0.086,Y -390.750,Z 1051.495,A 0.000,B 0.000,C 90.000,E1 269.141} C_DIS
LIN {X -0.067,Y -181.345,Z 1051.495,A 0.000,B 0.000,C 90.000,E1 269.141} C_DIS
LIN {X -0.009,Y -180.906,Z 1051.474,A 0.000,B 0.000,C 90.000,E1 265.412} C_DIS
LIN {X 0.047,Y -180.708,Z 1051.470,A 0.000,B 0.000,C 90.000,E1 264.552} C_DIS
LIN {X -0.034,Y -178.795,Z 1051.442,A 0.000,B 0.000,C 90.000,E1 259.511} C_DIS
LIN {X 0.042,Y -175.841,Z 1051.413,A 0.000,B 0.000,C 90.000,E1 254.393} C_DIS
LIN {X 0.042,Y -172.031,Z 1051.385,A 0.000,B 0.000,C 90.000,E1 249.263} C_DIS
LIN {X 0.018,Y -171.459,Z 1051.380,A 0.000,B 0.000,C 90.000,E1 248.411} C_DIS
LIN {X -0.001,Y -167.692,Z 1051.356,A 0.000,B 0.000,C 90.000,E1 244.101} C_DIS
LIN {X 0.012,Y -166.373,Z 1051.346,A 0.000,B 0.000,C 90.000,E1 242.359} C_DIS
LIN {X 0.004,Y -163.104,Z 1051.327,A 0.000,B 0.000,C 90.000,E1 238.869} C_DIS
LIN {X 0.054,Y -161.050,Z 1051.312,A 0.000,B 0.000,C 90.000,E1 236.215} C_DIS
LIN {X 0.037,Y -157.786,Z 1051.293,A 0.000,B 0.000,C 90.000,E1 232.683} C_DIS
LIN {X -0.019,Y -155.823,Z 1051.278,A 0.000,B 0.000,C 90.000,E1 230.033} C_DIS
LIN {X -0.062,Y -152.074,Z 1051.253,A 0.000,B 0.000,C 90.000,E1 225.567} C_DIS
LIN {X -0.043,Y -150.324,Z 1051.238,A 0.000,B 0.000,C 90.000,E1 222.852} C_DIS
LIN {X -0.020,Y -147.065,Z 1051.213,A 0.000,B 0.000,C 90.000,E1 218.302} C_DIS
LIN {X 0.086,Y -145.642,Z 1051.198,A 0.000,B 0.000,C 90.000,E1 215.518} C_DIS
LIN {X 0.084,Y -143.024,Z 1051.172,A 0.000,B 0.000,C 90.000,E1 210.924} C_DIS
LIN {X 0.015,Y -141.650,Z 1051.151,A 0.000,B 0.000,C 90.000,E1 207.257} C_DIS
LIN {X -0.065,Y -139.443,Z 1051.115,A 0.000,B 0.000,C 90.000,E1 200.791} C_DIS
LIN {X -0.013,Y -139.176,Z 1051.105,A 0.000,B 0.000,C 90.000,E1 198.906} C_DIS
LIN {X 0.015,Y -138.319,Z 1051.053,A 0.000,B 0.000,C 90.000,E1 189.557} C_DIS
LIN {X 0.024,Y -139.468,Z 1051.006,A 0.000,B 0.000,C 90.000,E1 181.146} C_DIS
LIN {X -0.035,Y -141.036,Z 1050.975,A 0.000,B 0.000,C 90.000,E1 175.584} C_DIS
LIN {X 0.060,Y -142.405,Z 1050.960,A 0.000,B 0.000,C 90.000,E1 172.761} C_DIS
LIN {X -0.018,Y -144.638,Z 1050.934,A 0.000,B 0.000,C 90.000,E1 168.173} C_DIS
LIN {X 0.041,Y -147.833,Z 1050.909,A 0.000,B 0.000,C 90.000,E1 163.559} C_DIS
LIN {X -0.014,Y -150.529,Z 1050.889,A 0.000,B 0.000,C 90.000,E1 159.934} C_DIS
LIN {X 0.005,Y -153.993,Z 1050.868,A 0.000,B 0.000,C 90.000,E1 156.305} C_DIS
LIN {X -0.075,Y -157.407,Z 1050.848,A 0.000,B 0.000,C 90.000,E1 152.743} C_DIS
LIN {X 0.005,Y -161.614,Z 1050.829,A 0.000,B 0.000,C 90.000,E1 149.154} C_DIS
LIN {X 0.107,Y -165.810,Z 1050.809,A 0.000,B 0.000,C 90.000,E1 145.595} C_DIS
LIN {X -0.004,Y -170.777,Z 1050.790,A 0.000,B 0.000,C 90.000,E1 142.145} C_DIS
LIN {X 0.017,Y -175.648,Z 1050.771,A 0.000,B 0.000,C 90.000,E1 138.690} C_DIS
LIN {X 0.015,Y -181.263,Z 1050.752,A 0.000,B 0.000,C 90.000,E1 135.283} C_DIS
LIN {X 0.016,Y -186.737,Z 1050.733,A 0.000,B 0.000,C 90.000,E1 131.919} C_DIS
LIN {X -0.033,Y -191.333,Z 1050.719,A 0.000,B 0.000,C 90.000,E1 129.439} C_DIS
LIN {X 0.036,Y -197.555,Z 1050.700,A 0.000,B 0.000,C 90.000,E1 125.931} C_DIS
LIN {X 0.014,Y -198.064,Z 1050.698,A 0.000,B 0.000,C 90.000,E1 125.678} C_DIS
LIN {X -0.039,Y -303.404,Z 1050.698,A 0.000,B 0.000,C 90.000,E1 125.678} C_DIS
LIN {X 0.078,Y -304.815,Z 1050.698,A 0.000,B 0.000,C 90.000,E1 125.644} C_DIS
LIN {X -0.138,Y -309.405,Z 1050.697,A 0.000,B 0.000,C 90.000,E1 125.518} C_DIS
LIN {X 0.077,Y -311.742,Z 1050.696,A 0.000,B 0.000,C 90.000,E1 125.311} C_DIS
LIN {X 0.007,Y -315.605,Z 1050.694,A 0.000,B 0.000,C 90.000,E1 124.898} C_DIS
LIN {X -0.079,Y -317.507,Z 1050.692,A 0.000,B 0.000,C 90.000,E1 124.612} C_DIS
LIN {X 0.096,Y -319.003,Z 1050.691,A 0.000,B 0.000,C 90.000,E1 124.278} C_DIS
LIN {X -0.024,Y -321.330,Z 1050.687,A 0.000,B 0.000,C 90.000,E1 123.658} C_DIS
LIN {X 0.023,Y -331.560,Z 1050.671,A 0.000,B 0.000,C 90.000,E1 120.797} C_DIS
LIN {X 0.139,Y -343.125,Z 1050.656,A 0.000,B 0.000,C 90.000,E1 117.975} C_DIS
LIN {X -0.197,Y -356.122,Z 1050.640,A 0.000,B 0.000,C 90.000,E1 115.283} C_DIS
LIN {X 0.102,Y -368.973,Z 1050.627,A 0.000,B 0.000,C 90.000,E1 112.845} C_DIS
LIN {X -0.108,Y -383.139,Z 1050.614,A 0.000,B 0.000,C 90.000,E1 110.536} C_DIS
LIN {X -0.027,Y -398.718,Z 1050.601,A 0.000,B 0.000,C 90.000,E1 108.236} C_DIS
LIN {X -0.178,Y -415.825,Z 1050.589,A 0.000,B 0.000,C 90.000,E1 106.024} C_DIS
LIN {X -0.020,Y -434.579,Z 1050.577,A 0.000,B 0.000,C 90.000,E1 103.828} C_DIS
LIN {X -0.034,Y -454.546,Z 1050.565,A 0.000,B 0.000,C 90.000,E1 101.771} C_DIS
LIN {X 0.156,Y -467.317,Z 1050.559,A 0.000,B 0.000,C 90.000,E1 100.546} C_DIS
LIN {X 0.159,Y -469.420,Z 1050.557,A 0.000,B 0.000,C 90.000,E1 100.310} C_DIS
LIN {X 0.161,Y -471.012,Z 1050.556,A 0.000,B 0.000,C 90.000,E1 100.074} C_DIS
LIN {X -0.066,Y -472.314,Z 1050.555,A 0.000,B 0.000,C 90.000,E1 99.849} C_DIS
LIN {X -0.214,Y -473.275,Z 1050.553,A 0.000,B 0.000,C 90.000,E1 99.613} C_DIS
LIN {X -0.103,Y -474.348,Z 1050.550,A 0.000,B 0.000,C 90.000,E1 99.095} C_DIS
LIN {X 0.089,Y -474.432,Z 1050.548,A 0.000,B 0.000,C 90.000,E1 98.568} C_DIS
LIN {X 0.215,Y -473.543,Z 1050.545,A 0.000,B 0.000,C 90.000,E1 98.049} C_DIS
LIN {X -0.126,Y -471.535,Z 1050.542,A 0.000,B 0.000,C 90.000,E1 97.587} C_DIS
LIN {X 0.199,Y -469.985,Z 1050.541,A 0.000,B 0.000,C 90.000,E1 97.296} C_DIS
LIN {X 0.055,Y -455.734,Z 1050.529,A 0.000,B 0.000,C 90.000,E1 95.277} C_DIS
LIN {X -0.090,Y -438.131,Z 1050.515,A 0.000,B 0.000,C 90.000,E1 92.694} C_DIS
LIN {X 0.036,Y -417.652,Z 1050.496,A 0.000,B 0.000,C 90.000,E1 89.198} C_DIS
LIN {X -0.073,Y -405.986,Z 1050.483,A 0.000,B 0.000,C 90.000,E1 87.020} C_DIS
LIN {X -0.108,Y -396.983,Z 1050.474,A 0.000,B 0.000,C 90.000,E1 85.355} C_DIS
LIN {X 0.123,Y -387.831,Z 1050.465,A 0.000,B 0.000,C 90.000,E1 83.628} C_DIS
LIN {X -0.147,Y -378.458,Z 1050.455,A 0.000,B 0.000,C 90.000,E1 81.951} C_DIS
LIN {X -0.145,Y -368.757,Z 1050.445,A 0.000,B 0.000,C 90.000,E1 80.208} C_DIS
LIN {X 0.033,Y -358.746,Z 1050.436,A 0.000,B 0.000,C 90.000,E1 78.409} C_DIS
LIN {X 0.101,Y -345.455,Z 1050.422,A 0.000,B 0.000,C 90.000,E1 75.992} C_DIS
LIN {X -0.179,Y -330.855,Z 1050.407,A 0.000,B 0.000,C 90.000,E1 73.268} C_DIS
LIN {X -0.087,Y -318.403,Z 1050.393,A 0.000,B 0.000,C 90.000,E1 70.732} C_DIS
LIN {X -0.083,Y -306.371,Z 1050.379,A 0.000,B 0.000,C 90.000,E1 68.156} C_DIS
LIN {X 0.129,Y -294.766,Z 1050.364,A 0.000,B 0.000,C 90.000,E1 65.485} C_DIS
LIN {X 0.017,Y -283.427,Z 1050.349,A 0.000,B 0.000,C 90.000,E1 62.820} C_DIS
LIN {X 0.015,Y -272.323,Z 1050.334,A 0.000,B 0.000,C 90.000,E1 60.078} C_DIS
LIN {X -0.123,Y -262.837,Z 1050.320,A 0.000,B 0.000,C 90.000,E1 57.661} C_DIS
LIN {X 0.080,Y -250.934,Z 1050.302,A 0.000,B 0.000,C 90.000,E1 54.402} C_DIS
LIN {X -0.149,Y -240.811,Z 1050.286,A 0.000,B 0.000,C 90.000,E1 51.537} C_DIS
LIN {X -0.057,Y -230.131,Z 1050.267,A 0.000,B 0.000,C 90.000,E1 48.162} C_DIS
LIN {X 0.098,Y -221.344,Z 1050.251,A 0.000,B 0.000,C 90.000,E1 45.081} C_DIS
LIN {X 0.055,Y -213.044,Z 1050.233,A 0.000,B 0.000,C 90.000,E1 42.000} C_DIS
LIN {X -0.022,Y -205.201,Z 1050.216,A 0.000,B 0.000,C 90.000,E1 38.874} C_DIS
LIN {X -0.032,Y -197.906,Z 1050.198,A 0.000,B 0.000,C 90.000,E1 35.678} C_DIS
LIN {X -0.005,Y -191.187,Z 1050.180,A 0.000,B 0.000,C 90.000,E1 32.418} C_DIS
LIN {X -0.031,Y -185.230,Z 1050.162,A 0.000,B 0.000,C 90.000,E1 29.127} C_DIS
LIN {X 0.008,Y -179.993,Z 1050.143,A 0.000,B 0.000,C 90.000,E1 25.771} C_DIS
LIN {X 0.012,Y -175.510,Z 1050.124,A 0.000,B 0.000,C 90.000,E1 22.386} C_DIS
LIN {X 0.036,Y -171.717,Z 1050.105,A 0.000,B 0.000,C 90.000,E1 18.960} C_DIS
LIN {X -0.010,Y -167.993,Z 1050.081,A 0.000,B 0.000,C 90.000,E1 14.662} C_DIS
LIN {X -0.004,Y -165.354,Z 1050.057,A 0.000,B 0.000,C 90.000,E1 10.310} C_DIS
LIN {X -0.071,Y -163.235,Z 1050.018,A 0.000,B 0.000,C 90.000,E1 3.326} C_DIS
LIN {X -0.033,Y -164.500,Z 1049.963,A 0.000,B 0.000,C 90.000,E1 353.394} C_DIS
LIN {X 0.049,Y -167.146,Z 1049.934,A 0.000,B 0.000,C 90.000,E1 348.117} C_DIS
LIN {X -0.019,Y -170.545,Z 1049.910,A 0.000,B 0.000,C 90.000,E1 343.795} C_DIS
LIN {X -0.096,Y -174.044,Z 1049.891,A 0.000,B 0.000,C 90.000,E1 340.369} C_DIS
LIN {X -0.019,Y -178.233,Z 1049.872,A 0.000,B 0.000,C 90.000,E1 336.922} C_DIS
LIN {X 0.051,Y -183.196,Z 1049.853,A 0.000,B 0.000,C 90.000,E1 333.512} C_DIS
LIN {X -0.086,Y -188.953,Z 1049.834,A 0.000,B 0.000,C 90.000,E1 330.205} C_DIS
LIN {X -0.026,Y -195.514,Z 1049.816,A 0.000,B 0.000,C 90.000,E1 326.882} C_DIS
LIN {X -0.015,Y -202.837,Z 1049.798,A 0.000,B 0.000,C 90.000,E1 323.623} C_DIS
LIN {X -0.039,Y -211.817,Z 1049.778,A 0.000,B 0.000,C 90.000,E1 320.033} C_DIS
LIN {X 0.002,Y -221.596,Z 1049.758,A 0.000,B 0.000,C 90.000,E1 316.500} C_DIS
LIN {X 0.053,Y -231.168,Z 1049.741,A 0.000,B 0.000,C 90.000,E1 313.419} C_DIS
LIN {X 0.072,Y -240.545,Z 1049.727,A 0.000,B 0.000,C 90.000,E1 310.782} C_DIS
LIN {X -0.031,Y -248.055,Z 1049.716,A 0.000,B 0.000,C 90.000,E1 308.955} C_DIS
LIN {X -0.160,Y -254.819,Z 1049.708,A 0.000,B 0.000,C 90.000,E1 307.523} C_DIS
LIN {X 0.009,Y -267.892,Z 1049.694,A 0.000,B 0.000,C 90.000,E1 304.978} C_DIS
LIN {X -0.149,Y -286.243,Z 1049.677,A 0.000,B 0.000,C 90.000,E1 301.878} C_DIS
LIN {X 0.021,Y -305.928,Z 1049.660,A 0.000,B 0.000,C 90.000,E1 298.821} C_DIS
LIN {X -0.026,Y -324.987,Z 1049.646,A 0.000,B 0.000,C 90.000,E1 296.232} C_DIS
LIN {X 0.168,Y -338.021,Z 1049.637,A 0.000,B 0.000,C 90.000,E1 294.643} C_DIS
LIN {X -0.053,Y -354.505,Z 1049.627,A 0.000,B 0.000,C 90.000,E1 292.950} C_DIS
LIN {X 0.163,Y -379.291,Z 1049.615,A 0.000,B 0.000,C 90.000,E1 290.610} C_DIS
LIN {X -0.097,Y -398.699,Z 1049.605,A 0.000,B 0.000,C 90.000,E1 288.960} C_DIS
LIN {X -0.031,Y -409.543,Z 1049.600,A 0.000,B 0.000,C 90.000,E1 288.000} C_DIS
LIN {X -0.023,Y -420.004,Z 1049.595,A 0.000,B 0.000,C 90.000,E1 287.040} C_DIS
LIN {X 0.167,Y -427.547,Z 1049.590,A 0.000,B 0.000,C 90.000,E1 286.260} C_DIS
LIN {X 0.198,Y -434.952,Z 1049.586,A 0.000,B 0.000,C 90.000,E1 285.481} C_DIS
LIN {X 0.137,Y -444.579,Z 1049.580,A 0.000,B 0.000,C 90.000,E1 284.426} C_DIS
LIN {X 0.062,Y -451.219,Z 1049.576,A 0.000,B 0.000,C 90.000,E1 283.647} C_DIS
LIN {X -0.074,Y -457.312,Z 1049.572,A 0.000,B 0.000,C 90.000,E1 282.883} C_DIS
LIN {X -0.152,Y -462.857,Z 1049.567,A 0.000,B 0.000,C 90.000,E1 282.119} C_DIS
LIN {X 0.268,Y -467.778,Z 1049.563,A 0.000,B 0.000,C 90.000,E1 281.299} C_DIS
LIN {X 0.192,Y -472.040,Z 1049.559,A 0.000,B 0.000,C 90.000,E1 280.546} C_DIS
LIN {X 0.155,Y -475.683,Z 1049.554,A 0.000,B 0.000,C 90.000,E1 279.792} C_DIS
LIN {X -0.112,Y -477.753,Z 1049.552,A 0.000,B 0.000,C 90.000,E1 279.321} C_DIS
LIN {X 0.026,Y -479.613,Z 1049.549,A 0.000,B 0.000,C 90.000,E1 278.803} C_DIS
LIN {X 0.243,Y -481.285,Z 1049.546,A 0.000,B 0.000,C 90.000,E1 278.276} C_DIS
LIN {X 0.094,Y -484.009,Z 1049.541,A 0.000,B 0.000,C 90.000,E1 277.296} C_DIS
LIN {X -0.209,Y -485.045,Z 1049.538,A 0.000,B 0.000,C 90.000,E1 276.834} C_DIS
LIN {X -0.022,Y -485.832,Z 1049.535,A 0.000,B 0.000,C 90.000,E1 276.315} C_DIS
LIN {X 0.172,Y -486.276,Z 1049.532,A 0.000,B 0.000,C 90.000,E1 275.796} C_DIS
LIN {X -0.117,Y -486.368,Z 1049.530,A 0.000,B 0.000,C 90.000,E1 275.334} C_DIS
LIN {X 0.041,Y -486.020,Z 1049.527,A 0.000,B 0.000,C 90.000,E1 274.821} C_DIS
LIN {X -0.244,Y -485.177,Z 1049.524,A 0.000,B 0.000,C 90.000,E1 274.359} C_DIS
LIN {X -0.049,Y -483.785,Z 1049.521,A 0.000,B 0.000,C 90.000,E1 273.841} C_DIS
LIN {X 0.109,Y -481.778,Z 1049.519,A 0.000,B 0.000,C 90.000,E1 273.326} C_DIS
LIN {X -0.193,Y -479.076,Z 1049.516,A 0.000,B 0.000,C 90.000,E1 272.865} C_DIS
LIN {X 0.112,Y -477.461,Z 1049.514,A 0.000,B 0.000,C 90.000,E1 272.579} C_DIS
LIN {X -0.237,Y -473.520,Z 1049.512,A 0.000,B 0.000,C 90.000,E1 272.121} C_DIS
LIN {X -0.114,Y -468.624,Z 1049.509,A 0.000,B 0.000,C 90.000,E1 271.604} C_DIS
LIN {X 0.135,Y -463.040,Z 1049.506,A 0.000,B 0.000,C 90.000,E1 271.088} C_DIS
LIN {X -0.194,Y -457.111,Z 1049.504,A 0.000,B 0.000,C 90.000,E1 270.688} C_DIS
LIN {X -0.143,Y -450.745,Z 1049.501,A 0.000,B 0.000,C 90.000,E1 270.286} C_DIS
LIN {X -0.115,Y -443.838,Z 1049.500,A 0.000,B 0.000,C 90.000,E1 269.943} C_DIS
LIN {X -0.035,Y -436.270,Z 1049.498,A 0.000,B 0.000,C 90.000,E1 269.656} C_DIS
LIN {X 0.124,Y -428.007,Z 1049.497,A 0.000,B 0.000,C 90.000,E1 269.427} C_DIS
LIN {X -0.102,Y -419.325,Z 1049.496,A 0.000,B 0.000,C 90.000,E1 269.312} C_DIS
LIN {X -0.011,Y -409.945,Z 1049.495,A 0.000,B 0.000,C 90.000,E1 269.198} C_DIS
LIN {X -0.028,Y -400.035,Z 1049.495,A 0.000,B 0.000,C 90.000,E1 269.141} C_DIS
LIN {X -0.139,Y -393.526,Z 1049.495,A 0.000,B 0.000,C 90.000,E1 269.141} C_DIS
LIN {X -0.089,Y -181.344,Z 1049.495,A 0.000,B 0.000,C 90.000,E1 269.141} C_DIS
LIN {X -0.081,Y -180.906,Z 1049.474,A 0.000,B 0.000,C 90.000,E1 265.412} C_DIS
LIN {X -0.007,Y -180.698,Z 1049.470,A 0.000,B 0.000,C 90.000,E1 264.546} C_DIS
LIN {X 0.071,Y -178.783,Z 1049.442,A 0.000,B 0.000,C 90.000,E1 259.454} C_DIS
LIN {X -0.028,Y -175.828,Z 1049.413,A 0.000,B 0.000,C 90.000,E1 254.393} C_DIS
LIN {X -0.027,Y -172.017,Z 1049.385,A 0.000,B 0.000,C 90.000,E1 249.263} C_DIS
LIN {X -0.050,Y -171.439,Z 1049.380,A 0.000,B 0.000,C 90.000,E1 248.411} C_DIS
LIN {X 0.004,Y -167.675,Z 1049.356,A 0.000,B 0.000,C 90.000,E1 244.076} C_DIS
LIN {X -0.055,Y -166.350,Z 1049.346,A 0.000,B 0.000,C 90.000,E1 242.359} C_DIS
LIN {X -0.063,Y -163.084,Z 1049.327,A 0.000,B 0.000,C 90.000,E1 238.869} C_DIS
LIN {X -0.012,Y -161.027,Z 1049.312,A 0.000,B 0.000,C 90.000,E1 236.215} C_DIS
LIN {X -0.028,Y -157.767,Z 1049.293,A 0.000,B 0.000,C 90.000,E1 232.683} C_DIS
LIN {X 0.035,Y -155.805,Z 1049.278,A 0.000,B 0.000,C 90.000,E1 229.989} C_DIS
LIN {X 0.090,Y -152.057,Z 1049.253,A 0.000,B 0.000,C 90.000,E1 225.486} C_DIS
LIN {X -0.004,Y -150.307,Z 1049.238,A 0.000,B 0.000,C 90.000,E1 222.813} C_DIS
LIN {X 0.032,Y -147.051,Z 1049.213,A 0.000,B 0.000,C 90.000,E1 218.257} C_DIS
LIN {X 0.024,Y -145.630,Z 1049.197,A 0.000,B 0.000,C 90.000,E1 215.518} C_DIS
LIN {X 0.023,Y -143.013,Z 1049.172,A 0.000,B 0.000,C 90.000,E1 210.924} C_DIS
LIN {X -0.046,Y -141.639,Z 1049.151,A 0.000,B 0.000,C 90.000,E1 207.257} C_DIS
LIN {X 0.005,Y -139.438,Z 1049.115,A 0.000,B 0.000,C 90.000,E1 200.737} C_DIS
LIN {X -0.074,Y -139.171,Z 1049.105,A 0.000,B 0.000,C 90.000,E1 198.906} C_DIS
LIN {X -0.045,Y -138.317,Z 1049.053,A 0.000,B 0.000,C 90.000,E1 189.557} C_DIS
LIN {X -0.036,Y -139.472,Z 1049.006,A 0.000,B 0.000,C 90.000,E1 181.146} C_DIS
LIN {X 0.044,Y -141.047,Z 1048.975,A 0.000,B 0.000,C 90.000,E1 175.527} C_DIS
LIN {X -0.001,Y -142.418,Z 1048.960,A 0.000,B 0.000,C 90.000,E1 172.761} C_DIS
LIN {X 0.061,Y -144.653,Z 1048.934,A 0.000,B 0.000,C 90.000,E1 168.117} C_DIS
LIN {X -0.022,Y -147.850,Z 1048.909,A 0.000,B 0.000,C 90.000,E1 163.559} C_DIS
LIN {X 0.064,Y -150.550,Z 1048.888,A 0.000,B 0.000,C 90.000,E1 159.880} C_DIS
LIN {X -0.060,Y -154.016,Z 1048.868,A 0.000,B 0.000,C 90.000,E1 156.305} C_DIS
LIN {X 0.000,Y -157.431,Z 1048.848,A 0.000,B 0.000,C 90.000,E1 152.692} C_DIS
LIN {X 0.021,Y -161.644,Z 1048.828,A 0.000,B 0.000,C 90.000,E1 149.125} C_DIS
LIN {X 0.039,Y -165.841,Z 1048.809,A 0.000,B 0.000,C 90.000,E1 145.595} C_DIS
LIN {X 0.031,Y -170.813,Z 1048.790,A 0.000,B 0.000,C 90.000,E1 142.110} C_DIS
LIN {X -0.053,Y -175.682,Z 1048.770,A 0.000,B 0.000,C 90.000,E1 138.690} C_DIS
LIN {X 0.071,Y -181.296,Z 1048.751,A 0.000,B 0.000,C 90.000,E1 135.243} C_DIS
LIN {X -0.057,Y -186.776,Z 1048.733,A 0.000,B 0.000,C 90.000,E1 131.919} C_DIS
LIN {X 0.015,Y -191.369,Z 1048.719,A 0.000,B 0.000,C 90.000,E1 129.402} C_DIS
LIN {X -0.037,Y -197.596,Z 1048.700,A 0.000,B 0.000,C 90.000,E1 125.931} C_DIS
LIN {X -0.028,Y -197.997,Z 1048.698,A 0.000,B 0.000,C 90.000,E1 125.724} C_DIS
LIN {X -0.078,Y -303.752,Z 1048.698,A 0.000,B 0.000,C 90.000,E1 125.724} C_DIS
LIN {X 0.034,Y -305.537,Z 1048.698,A 0.000,B 0.000,C 90.000,E1 125.678} C_DIS
LIN {X -0.130,Y -309.891,Z 1048.697,A 0.000,B 0.000,C 90.000,E1 125.518} C_DIS
LIN {X -0.041,Y -312.298,Z 1048.696,A 0.000,B 0.000,C 90.000,E1 125.311} C_DIS
LIN {X 0.114,Y -316.145,Z 1048.694,A 0.000,B 0.000,C 90.000,E1 124.818} C_DIS
LIN {X -0.084,Y -317.995,Z 1048.692,A 0.000,B 0.000,C 90.000,E1 124.532} C_DIS
LIN {X -0.021,Y -319.441,Z 1048.690,A 0.000,B 0.000,C 90.000,E1 124.199} C_DIS
LIN {X -0.092,Y -331.918,Z 1048.671,A 0.000,B 0.000,C 90.000,E1 120.718} C_DIS
LIN {X 0.024,Y -343.532,Z 1048.655,A 0.000,B 0.000,C 90.000,E1 117.897} C_DIS
LIN {X 0.010,Y -356.580,Z 1048.640,A 0.000,B 0.000,C 90.000,E1 115.155} C_DIS
LIN {X -0.013,Y -369.480,Z 1048.626,A 0.000,B 0.000,C 90.000,E1 112.770} C_DIS
LIN {X 0.000,Y -383.700,Z 1048.614,A 0.000,B 0.000,C 90.000,E1 110.429} C_DIS
LIN {X 0.112,Y -399.337,Z 1048.601,A 0.000,B 0.000,C 90.000,E1 108.127} C_DIS
LIN {X 0.105,Y -416.505,Z 1048.588,A 0.000,B 0.000,C 90.000,E1 105.898} C_DIS
LIN {X -0.240,Y -435.326,Z 1048.576,A 0.000,B 0.000,C 90.000,E1 103.772} C_DIS
LIN {X -0.210,Y -455.324,Z 1048.565,A 0.000,B 0.000,C 90.000,E1 101.715} C_DIS
LIN {X 0.010,Y -468.021,Z 1048.558,A 0.000,B 0.000,C 90.000,E1 100.489} C_DIS
LIN {X -0.023,Y -469.975,Z 1048.557,A 0.000,B 0.000,C 90.000,E1 100.254} C_DIS
LIN {X -0.058,Y -471.459,Z 1048.556,A 0.000,B 0.000,C 90.000,E1 100.018} C_DIS
LIN {X 0.262,Y -472.643,Z 1048.554,A 0.000,B 0.000,C 90.000,E1 99.726} C_DIS
LIN {X 0.038,Y -473.505,Z 1048.553,A 0.000,B 0.000,C 90.000,E1 99.500} C_DIS
LIN {X 0.227,Y -474.412,Z 1048.550,A 0.000,B 0.000,C 90.000,E1 98.973} C_DIS
LIN {X -0.122,Y -474.343,Z 1048.547,A 0.000,B 0.000,C 90.000,E1 98.511} C_DIS
LIN {X 0.005,Y -473.289,Z 1048.544,A 0.000,B 0.000,C 90.000,E1 97.992} C_DIS
LIN {X -0.133,Y -472.347,Z 1048.543,A 0.000,B 0.000,C 90.000,E1 97.757} C_DIS
LIN {X 0.133,Y -471.071,Z 1048.542,A 0.000,B 0.000,C 90.000,E1 97.473} C_DIS
LIN {X 0.014,Y -460.474,Z 1048.533,A 0.000,B 0.000,C 90.000,E1 95.967} C_DIS
LIN {X 0.074,Y -449.759,Z 1048.525,A 0.000,B 0.000,C 90.000,E1 94.416} C_DIS
LIN {X -0.143,Y -435.942,Z 1048.513,A 0.000,B 0.000,C 90.000,E1 92.350} C_DIS
LIN {X -0.199,Y -417.141,Z 1048.495,A 0.000,B 0.000,C 90.000,E1 89.141} C_DIS
LIN {X 0.022,Y -406.975,Z 1048.484,A 0.000,B 0.000,C 90.000,E1 87.192} C_DIS
LIN {X 0.005,Y -398.005,Z 1048.475,A 0.000,B 0.000,C 90.000,E1 85.527} C_DIS
